LIN {X 0,Y 137.827,Z 379.001,A -85,B 0,C 180,E1 -25699.087,E2 -25699.087} C_VEL
LIN {X 0,Y 133.613,Z 369.148,A -85,B 0,C 180,E1 -25701.525,E2 -25701.525} C_VEL
LIN {X 0,Y 127.803,Z 359.632,A -85,B 0,C 180,E1 -25704.98,E2 -25704.98} C_VEL
LIN {X 0,Y 124.55,Z 355.02,A -85,B 0,C 180,E1 -25707.103,E2 -25707.103} C_VEL
LIN {X 0,Y 121.893,Z 351.23,A -85,B 0,C 180,E1 -25709.002,E2 -25709.002} C_VEL
LIN {X 0,Y 119.524,Z 348.351,A -85,B 0,C 180,E1 -25710.791,E2 -25710.791} C_VEL
LIN {X 0,Y 118.503,Z 346.486,A -85,B 0,C 180,E1 -25711.675,E2 -25711.675} C_VEL
LIN {X 0,Y 116.133,Z 344.433,A -85,B 0,C 180,E1 -25713.613,E2 -25713.613} C_VEL
LIN {X 0,Y 115.029,Z 342.02,A -85,B 0,C 180,E1 -25714.749,E2 -25714.749} C_VEL
LIN {X 0,Y 114.889,Z 341.174,A -85,B 0,C 180,E1 -25715.069,E2 -25715.069} C_VEL
LIN {X 0,Y 114.953,Z 341.137,A -85,B 0,C 180,E1 -25718.479,E2 -25718.479} C_VEL
LIN {X 0,Y 115.104,Z 341.145,A -85,B 0,C 180,E1 -25725.863,E2 -25725.863} C_VEL
LIN {X 0,Y 115.312,Z 341.081,A -85,B 0,C 180,E1 -25729.464,E2 -25729.464} C_VEL
LIN {X 0,Y 115.511,Z 341.094,A -85,B 0,C 180,E1 -25736.511,E2 -25736.511} C_VEL
LIN {X 0,Y 115.983,Z 341.003,A -85,B 0,C 180,E1 -25739.999,E2 -25739.999} C_VEL
LIN {X 0,Y 115.359,Z 341.105,A -85,B 0,C 180,E1 -25746.998,E2 -25746.998} C_VEL
LIN {X 0,Y 115.21,Z 341.099,A -85,B 0,C 180,E1 -25752.558,E2 -25752.558} C_VEL
LIN {X 0,Y 114.973,Z 341.127,A -85,B 0,C 180,E1 -25757.796,E2 -25757.796} C_VEL
LIN {X 0,Y 114.926,Z 341.156,A -85,B 0,C 180,E1 -25763.461,E2 -25763.461} C_VEL
LIN {X 0,Y 114.858,Z 341.154,A -85,B 0,C 180,E1 -25771.054,E2 -25771.054} C_VEL
LIN {X 0,Y 114.778,Z 341.146,A -85,B 0,C 180,E1 -25777.756,E2 -25777.756} C_VEL
LIN {X 0,Y 114.822,Z 341.142,A -85,B 0,C 180,E1 -25779.421,E2 -25779.421} C_VEL
LIN {X 0,Y 115.614,Z 343.676,A -85,B 0,C 180,E1 -25780.373,E2 -25780.373} C_VEL
LIN {X 0,Y 117.731,Z 346.081,A -85,B 0,C 180,E1 -25782.211,E2 -25782.211} C_VEL
LIN {X 0,Y 118.812,Z 346.913,A -85,B 0,C 180,E1 -25783.051,E2 -25783.051} C_VEL
LIN {X 0,Y 120.793,Z 350.186,A -85,B 0,C 180,E1 -25784.683,E2 -25784.683} C_VEL
LIN {X 0,Y 122.393,Z 351.931,A -85,B 0,C 180,E1 -25785.836,E2 -25785.836} C_VEL
LIN {X 0,Y 125.131,Z 355.737,A -85,B 0,C 180,E1 -25787.75,E2 -25787.75} C_VEL
LIN {X 0,Y 131.366,Z 365.259,A -85,B 0,C 180,E1 -25791.647,E2 -25791.647} C_VEL
LIN {X 0,Y 135.538,Z 372.511,A -85,B 0,C 180,E1 -25793.998,E2 -25793.998} C_VEL
LIN {X 0,Y 140.144,Z 381.658,A -85,B 0,C 180,E1 -25796.428,E2 -25796.428} C_VEL
LIN {X 0,Y 143.275,Z 388.687,A -85,B 0,C 180,E1 -25797.995,E2 -25797.995} C_VEL
LIN {X 0,Y 142.115,Z 408.083,A -85,B 0,C 180,E1 -25798.87,E2 -25798.87} C_VEL
LIN {X 0,Y 139.875,Z 437.734,A -85,B 0,C 180,E1 -25800.177,E2 -25800.177} C_VEL
LIN {X 0,Y 138.032,Z 451.323,A -85,B 0,C 180,E1 -25801.289,E2 -25801.289} C_VEL
LIN {X 0,Y 135.673,Z 463.657,A -85,B 0,C 180,E1 -25802.836,E2 -25802.836} C_VEL
LIN {X 0,Y 132.815,Z 475.522,A -85,B 0,C 180,E1 -25804.952,E2 -25804.952} C_VEL
LIN {X 0,Y 129.446,Z 486.941,A -85,B 0,C 180,E1 -25807.66,E2 -25807.66} C_VEL
LIN {X 0,Y 125.81,Z 497.272,A -85,B 0,C 180,E1 -25810.838,E2 -25810.838} C_VEL
LIN {X 0,Y 121.985,Z 507.34,A -85,B 0,C 180,E1 -25814.971,E2 -25814.971} C_VEL
LIN {X 0,Y 118.496,Z 516.2,A -85,B 0,C 180,E1 -25819.748,E2 -25819.748} C_VEL
LIN {X 0,Y 115.779,Z 523.275,A -85,B 0,C 180,E1 -25824.773,E2 -25824.773} C_VEL
LIN {X 0,Y 113.838,Z 528.929,A -85,B 0,C 180,E1 -25829.997,E2 -25829.997} C_VEL
LIN {X 0,Y 112.806,Z 532.82,A -85,B 0,C 180,E1 -25834.575,E2 -25834.575} C_VEL
LIN {X 0,Y 111.862,Z 536.768,A -85,B 0,C 180,E1 -25840.861,E2 -25840.861} C_VEL
LIN {X 0,Y 111.797,Z 538.454,A -85,B 0,C 180,E1 -25844.56,E2 -25844.56} C_VEL
LIN {X 0,Y 112.379,Z 540.208,A -85,B 0,C 180,E1 -25850.271,E2 -25850.271} C_VEL
LIN {X 0,Y 113.544,Z 540.951,A -85,B 0,C 180,E1 -25855.672,E2 -25855.672} C_VEL
LIN {X 0,Y 116.294,Z 540.626,A -85,B 0,C 180,E1 -25862.216,E2 -25862.216} C_VEL
LIN {X 0,Y 118.676,Z 539.642,A -85,B 0,C 180,E1 -25866.309,E2 -25866.309} C_VEL
LIN {X 0,Y 123.502,Z 536.925,A -85,B 0,C 180,E1 -25872.289,E2 -25872.289} C_VEL
LIN {X 0,Y 129.003,Z 533.061,A -85,B 0,C 180,E1 -25877.342,E2 -25877.342} C_VEL
LIN {X 0,Y 134.673,Z 528.328,A -85,B 0,C 180,E1 -25881.511,E2 -25881.511} C_VEL
LIN {X 0,Y 140.964,Z 522.244,A -85,B 0,C 180,E1 -25885.345,E2 -25885.345} C_VEL
LIN {X 0,Y 147.922,Z 514.608,A -85,B 0,C 180,E1 -25888.777,E2 -25888.777} C_VEL
LIN {X 0,Y 154.047,Z 506.758,A -85,B 0,C 180,E1 -25891.424,E2 -25891.424} C_VEL
LIN {X 0,Y 160.683,Z 496.79,A -85,B 0,C 180,E1 -25893.929,E2 -25893.929} C_VEL
LIN {X 0,Y 166.481,Z 486.303,A -85,B 0,C 180,E1 -25895.903,E2 -25895.903} C_VEL
LIN {X 0,Y 171.312,Z 475.836,A -85,B 0,C 180,E1 -25897.37,E2 -25897.37} C_VEL
LIN {X 0,Y 175.536,Z 464.261,A -85,B 0,C 180,E1 -25898.628,E2 -25898.628} C_VEL
LIN {X 0,Y 178.99,Z 451.384,A -85,B 0,C 180,E1 -25899.64,E2 -25899.64} C_VEL
LIN {X 0,Y 181.472,Z 437.921,A -85,B 0,C 180,E1 -25900.311,E2 -25900.311} C_VEL
LIN {X 0,Y 183.082,Z 422.653,A -85,B 0,C 180,E1 -25900.76,E2 -25900.76} C_VEL
LIN {X 0,Y 179.542,Z 415.553,A -85,B 0,C 180,E1 -25903.806,E2 -25903.806} C_VEL
LIN {X 0,Y 176.526,Z 410.032,A -85,B 0,C 180,E1 -25906.785,E2 -25906.785} C_VEL
LIN {X 0,Y 174.132,Z 405.888,A -85,B 0,C 180,E1 -25909.54,E2 -25909.54} C_VEL
LIN {X 0,Y 172.909,Z 403.751,A -85,B 0,C 180,E1 -25911.158,E2 -25911.158} C_VEL
LIN {X 0,Y 170.704,Z 399.785,A -85,B 0,C 180,E1 -25914.759,E2 -25914.759} C_VEL
LIN {X 0,Y 168.841,Z 396.541,A -85,B 0,C 180,E1 -25919.062,E2 -25919.062} C_VEL
LIN {X 0,Y 168.584,Z 395.7,A -85,B 0,C 180,E1 -25920.001,E2 -25920.001} C_VEL
LIN {X 0,Y 167.507,Z 395.197,A -85,B 0,C 180,E1 -25924.814,E2 -25924.814} C_VEL
LIN {X 0,Y 167.607,Z 395.272,A -85,B 0,C 180,E1 -25929.656,E2 -25929.656} C_VEL
LIN {X 0,Y 168.546,Z 396.155,A -85,B 0,C 180,E1 -25933.716,E2 -25933.716} C_VEL
LIN {X 0,Y 170.103,Z 399.496,A -85,B 0,C 180,E1 -25937.876,E2 -25937.876} C_VEL
LIN {X 0,Y 171.176,Z 400.958,A -85,B 0,C 180,E1 -25939.832,E2 -25939.832} C_VEL
LIN {X 0,Y 173.514,Z 405.486,A -85,B 0,C 180,E1 -25943.419,E2 -25943.419} C_VEL
LIN {X 0,Y 175.851,Z 410.567,A -85,B 0,C 180,E1 -25946.348,E2 -25946.348} C_VEL
LIN {X 0,Y 178.897,Z 417.775,A -85,B 0,C 180,E1 -25949.606,E2 -25949.606} C_VEL
LIN {X 0,Y 181.846,Z 425.459,A -85,B 0,C 180,E1 -25952.37,E2 -25952.37} C_VEL
LIN {X 0,Y 182.641,Z 427.679,A -85,B 0,C 180,E1 -25953.068,E2 -25953.068} C_VEL
LIN {X 0,Y 180.767,Z 445.11,A -85,B 0,C 180,E1 -25953.661,E2 -25953.661} C_VEL
LIN {X 0,Y 178.134,Z 458.354,A -85,B 0,C 180,E1 -25954.359,E2 -25954.359} C_VEL
LIN {X 0,Y 174.747,Z 469.708,A -85,B 0,C 180,E1 -25955.168,E2 -25955.168} C_VEL
LIN {X 0,Y 170.165,Z 481.545,A -85,B 0,C 180,E1 -25956.358,E2 -25956.358} C_VEL
LIN {X 0,Y 164.843,Z 492.752,A -85,B 0,C 180,E1 -25957.936,E2 -25957.936} C_VEL
LIN {X 0,Y 158.973,Z 502.9,A -85,B 0,C 180,E1 -25959.818,E2 -25959.818} C_VEL
LIN {X 0,Y 153.372,Z 511.22,A -85,B 0,C 180,E1 -25961.877,E2 -25961.877} C_VEL
LIN {X 0,Y 146.218,Z 520.28,A -85,B 0,C 180,E1 -25964.853,E2 -25964.853} C_VEL
LIN {X 0,Y 139.495,Z 527.609,A -85,B 0,C 180,E1 -25968.125,E2 -25968.125} C_VEL
LIN {X 0,Y 134.368,Z 532.602,A -85,B 0,C 180,E1 -25971.127,E2 -25971.127} C_VEL
LIN {X 0,Y 129.267,Z 537.189,A -85,B 0,C 180,E1 -25974.823,E2 -25974.823} C_VEL
LIN {X 0,Y 124.031,Z 541.242,A -85,B 0,C 180,E1 -25979.342,E2 -25979.342} C_VEL
LIN {X 0,Y 118.724,Z 544.762,A -85,B 0,C 180,E1 -25985.524,E2 -25985.524} C_VEL
LIN {X 0,Y 116.569,Z 545.891,A -85,B 0,C 180,E1 -25988.796,E2 -25988.796} C_VEL
LIN {X 0,Y 113.713,Z 546.98,A -85,B 0,C 180,E1 -25995.69,E2 -25995.69} C_VEL
LIN {X 0,Y 112.862,Z 546.963,A -85,B 0,C 180,E1 -25999.237,E2 -25999.237} C_VEL
LIN {X 0,Y 112.354,Z 546.555,A -85,B 0,C 180,E1 -26002.817,E2 -26002.817} C_VEL
LIN {X 0,Y 112.262,Z 545.725,A -85,B 0,C 180,E1 -26006.414,E2 -26006.414} C_VEL
LIN {X 0,Y 112.334,Z 544.497,A -85,B 0,C 180,E1 -26010.003,E2 -26010.003} C_VEL
LIN {X 0,Y 112.247,Z 541.82,A -85,B 0,C 180,E1 -26015.392,E2 -26015.392} C_VEL
LIN {X 0,Y 112.798,Z 538.095,A -85,B 0,C 180,E1 -26020.776,E2 -26020.776} C_VEL
LIN {X 0,Y 113.999,Z 533.213,A -85,B 0,C 180,E1 -26026.11,E2 -26026.11} C_VEL
LIN {X 0,Y 116.159,Z 527.043,A -85,B 0,C 180,E1 -26031.289,E2 -26031.289} C_VEL
LIN {X 0,Y 119.107,Z 519.342,A -85,B 0,C 180,E1 -26036.269,E2 -26036.269} C_VEL
LIN {X 0,Y 122.141,Z 511.23,A -85,B 0,C 180,E1 -26040.332,E2 -26040.332} C_VEL
LIN {X 0,Y 125.723,Z 501.735,A -85,B 0,C 180,E1 -26043.99,E2 -26043.99} C_VEL
LIN {X 0,Y 129.315,Z 490.95,A -85,B 0,C 180,E1 -26047.205,E2 -26047.205} C_VEL
LIN {X 0,Y 132.655,Z 480.586,A -85,B 0,C 180,E1 -26049.479,E2 -26049.479} C_VEL
LIN {X 0,Y 133.738,Z 476.295,A -85,B 0,C 180,E1 -26050.286,E2 -26050.286} C_VEL
LIN {X 0,Y 134.047,Z 472.751,A -85,B 0,C 180,E1 -26051.07,E2 -26051.07} C_VEL
LIN {X 0,Y 132.999,Z 467.14,A -85,B 0,C 180,E1 -26052.639,E2 -26052.639} C_VEL
LIN {X 0,Y 131.908,Z 461.392,A -85,B 0,C 180,E1 -26054.093,E2 -26054.093} C_VEL
LIN {X 0,Y 132.097,Z 457.639,A -85,B 0,C 180,E1 -26054.66,E2 -26054.66} C_VEL
LIN {X 0,Y 134.126,Z 443.975,A -85,B 0,C 180,E1 -26055.786,E2 -26055.786} C_VEL
LIN {X 0,Y 137.136,Z 402.806,A -85,B 0,C 180,E1 -26057.681,E2 -26057.681} C_VEL
LIN {X 0,Y 137.217,Z 397.25,A -85,B 0,C 180,E1 -26058.038,E2 -26058.038} C_VEL
LIN {X 0,Y 136.74,Z 393.549,A -85,B 0,C 180,E1 -26058.476,E2 -26058.476} C_VEL
LIN {X 0,Y 132.767,Z 381.798,A -85,B 0,C 180,E1 -26060.93,E2 -26060.93} C_VEL
LIN {X 0,Y 129.383,Z 373.685,A -85,B 0,C 180,E1 -26063.064,E2 -26063.064} C_VEL
LIN {X 0,Y 123.95,Z 364.6,A -85,B 0,C 180,E1 -26066.572,E2 -26066.572} C_VEL
LIN {X 0,Y 118.97,Z 357.189,A -85,B 0,C 180,E1 -26070.254,E2 -26070.254} C_VEL
LIN {X 0,Y 116.317,Z 353.693,A -85,B 0,C 180,E1 -26072.444,E2 -26072.444} C_VEL
LIN {X 0,Y 115.584,Z 352.531,A -85,B 0,C 180,E1 -26073.112,E2 -26073.112} C_VEL
LIN {X 0,Y 113.146,Z 349.883,A -85,B 0,C 180,E1 -26075.342,E2 -26075.342} C_VEL
LIN {X 0,Y 112.083,Z 347.678,A -85,B 0,C 180,E1 -26076.525,E2 -26076.525} C_VEL
LIN {X 0,Y 109.323,Z 345.51,A -85,B 0,C 180,E1 -26079.416,E2 -26079.416} C_VEL
LIN {X 0,Y 108.116,Z 343.183,A -85,B 0,C 180,E1 -26081.032,E2 -26081.032} C_VEL
LIN {X 0,Y 107.892,Z 342.014,A -85,B 0,C 180,E1 -26081.484,E2 -26081.484} C_VEL
LIN {X 0,Y 108.212,Z 341.969,A -85,B 0,C 180,E1 -26088.764,E2 -26088.764} C_VEL
LIN {X 0,Y 108.296,Z 341.957,A -85,B 0,C 180,E1 -26092.542,E2 -26092.542} C_VEL
LIN {X 0,Y 108.909,Z 341.882,A -85,B 0,C 180,E1 -26099.999,E2 -26099.999} C_VEL
LIN {X 0,Y 108.298,Z 341.987,A -85,B 0,C 180,E1 -26107.457,E2 -26107.457} C_VEL
LIN {X 0,Y 108.144,Z 341.974,A -85,B 0,C 180,E1 -26112.873,E2 -26112.873} C_VEL
LIN {X 0,Y 107.872,Z 342.025,A -85,B 0,C 180,E1 -26119.01,E2 -26119.01} C_VEL
LIN {X 0,Y 107.833,Z 342.028,A -85,B 0,C 180,E1 -26124.147,E2 -26124.147} C_VEL
LIN {X 0,Y 107.765,Z 342.055,A -85,B 0,C 180,E1 -26132.742,E2 -26132.742} C_VEL
LIN {X 0,Y 108.751,Z 344.913,A -85,B 0,C 180,E1 -26134.366,E2 -26134.366} C_VEL
LIN {X 0,Y 110.78,Z 347.032,A -85,B 0,C 180,E1 -26136.674,E2 -26136.674} C_VEL
LIN {X 0,Y 112.145,Z 347.931,A -85,B 0,C 180,E1 -26138.028,E2 -26138.028} C_VEL
LIN {X 0,Y 113.954,Z 351.053,A -85,B 0,C 180,E1 -26139.925,E2 -26139.925} C_VEL
LIN {X 0,Y 116.048,Z 353.188,A -85,B 0,C 180,E1 -26141.771,E2 -26141.771} C_VEL
LIN {X 0,Y 118.459,Z 356.701,A -85,B 0,C 180,E1 -26143.827,E2 -26143.827} C_VEL
LIN {X 0,Y 119.687,Z 358.436,A -85,B 0,C 180,E1 -26144.799,E2 -26144.799} C_VEL
LIN {X 0,Y 123.602,Z 364.137,A -85,B 0,C 180,E1 -26147.66,E2 -26147.66} C_VEL
LIN {X 0,Y 128.584,Z 372.074,A -85,B 0,C 180,E1 -26150.898,E2 -26150.898} C_VEL
LIN {X 0,Y 134.41,Z 383.213,A -85,B 0,C 180,E1 -26154.323,E2 -26154.323} C_VEL
LIN {X 0,Y 137.862,Z 391.022,A -85,B 0,C 180,E1 -26156.231,E2 -26156.231} C_VEL
LIN {X 0,Y 134.356,Z 437.827,A -85,B 0,C 180,E1 -26158.318,E2 -26158.318} C_VEL
LIN {X 0,Y 132.383,Z 451.784,A -85,B 0,C 180,E1 -26159.489,E2 -26159.489} C_VEL
LIN {X 0,Y 129.88,Z 464.097,A -85,B 0,C 180,E1 -26161.075,E2 -26161.075} C_VEL
LIN {X 0,Y 126.877,Z 475.904,A -85,B 0,C 180,E1 -26163.249,E2 -26163.249} C_VEL
LIN {X 0,Y 123.326,Z 487.32,A -85,B 0,C 180,E1 -26166.052,E2 -26166.052} C_VEL
LIN {X 0,Y 119.5,Z 497.588,A -85,B 0,C 180,E1 -26169.334,E2 -26169.334} C_VEL
LIN {X 0,Y 115.821,Z 506.81,A -85,B 0,C 180,E1 -26173.245,E2 -26173.245} C_VEL
LIN {X 0,Y 112.034,Z 515.794,A -85,B 0,C 180,E1 -26178.233,E2 -26178.233} C_VEL
LIN {X 0,Y 109.056,Z 523.018,A -85,B 0,C 180,E1 -26183.521,E2 -26183.521} C_VEL
LIN {X 0,Y 107.232,Z 527.89,A -85,B 0,C 180,E1 -26188.119,E2 -26188.119} C_VEL
LIN {X 0,Y 105.721,Z 533.01,A -85,B 0,C 180,E1 -26194.334,E2 -26194.334} C_VEL
LIN {X 0,Y 104.888,Z 536.261,A -85,B 0,C 180,E1 -26199.64,E2 -26199.64} C_VEL
LIN {X 0,Y 104.732,Z 538.867,A -85,B 0,C 180,E1 -26205.567,E2 -26205.567} C_VEL
LIN {X 0,Y 105.375,Z 540.383,A -85,B 0,C 180,E1 -26210.978,E2 -26210.978} C_VEL
LIN {X 0,Y 106.907,Z 541.182,A -85,B 0,C 180,E1 -26217.394,E2 -26217.394} C_VEL
LIN {X 0,Y 109.666,Z 540.852,A -85,B 0,C 180,E1 -26223.582,E2 -26223.582} C_VEL
LIN {X 0,Y 112.772,Z 539.685,A -85,B 0,C 180,E1 -26228.546,E2 -26228.546} C_VEL
LIN {X 0,Y 117.499,Z 537.203,A -85,B 0,C 180,E1 -26234.131,E2 -26234.131} C_VEL
LIN {X 0,Y 122.194,Z 534.189,A -85,B 0,C 180,E1 -26238.386,E2 -26238.386} C_VEL
LIN {X 0,Y 128.546,Z 529.387,A -85,B 0,C 180,E1 -26243.03,E2 -26243.03} C_VEL
LIN {X 0,Y 135.72,Z 522.973,A -85,B 0,C 180,E1 -26247.291,E2 -26247.291} C_VEL
LIN {X 0,Y 142.801,Z 515.651,A -85,B 0,C 180,E1 -26250.67,E2 -26250.67} C_VEL
LIN {X 0,Y 149.335,Z 507.74,A -85,B 0,C 180,E1 -26253.397,E2 -26253.397} C_VEL
LIN {X 0,Y 156.111,Z 498.172,A -85,B 0,C 180,E1 -26255.846,E2 -26255.846} C_VEL
LIN {X 0,Y 162.206,Z 487.75,A -85,B 0,C 180,E1 -26257.832,E2 -26257.832} C_VEL
LIN {X 0,Y 167.172,Z 477.558,A -85,B 0,C 180,E1 -26259.286,E2 -26259.286} C_VEL
LIN {X 0,Y 172.029,Z 464.986,A -85,B 0,C 180,E1 -26260.649,E2 -26260.649} C_VEL
LIN {X 0,Y 175.423,Z 453.15,A -85,B 0,C 180,E1 -26261.583,E2 -26261.583} C_VEL
LIN {X 0,Y 178.092,Z 439.722,A -85,B 0,C 180,E1 -26262.267,E2 -26262.267} C_VEL
LIN {X 0,Y 179.652,Z 426.224,A -85,B 0,C 180,E1 -26262.69,E2 -26262.69} C_VEL
LIN {X 0,Y 176.367,Z 419.516,A -85,B 0,C 180,E1 -26265.851,E2 -26265.851} C_VEL
LIN {X 0,Y 173.495,Z 414.015,A -85,B 0,C 180,E1 -26269.106,E2 -26269.106} C_VEL
LIN {X 0,Y 171.402,Z 410.289,A -85,B 0,C 180,E1 -26271.942,E2 -26271.942} C_VEL
LIN {X 0,Y 169.34,Z 406.418,A -85,B 0,C 180,E1 -26275.593,E2 -26275.593} C_VEL
LIN {X 0,Y 167.703,Z 403.164,A -85,B 0,C 180,E1 -26279.843,E2 -26279.843} C_VEL
LIN {X 0,Y 167.333,Z 402.501,A -85,B 0,C 180,E1 -26281.204,E2 -26281.204} C_VEL
LIN {X 0,Y 166.57,Z 402.195,A -85,B 0,C 180,E1 -26288.143,E2 -26288.143} C_VEL
LIN {X 0,Y 167.549,Z 403.229,A -85,B 0,C 180,E1 -26293.411,E2 -26293.411} C_VEL
LIN {X 0,Y 169.1,Z 406.549,A -85,B 0,C 180,E1 -26297.693,E2 -26297.693} C_VEL
LIN {X 0,Y 169.95,Z 407.804,A -85,B 0,C 180,E1 -26299.32,E2 -26299.32} C_VEL
LIN {X 0,Y 171.934,Z 412,A -85,B 0,C 180,E1 -26302.613,E2 -26302.613} C_VEL
LIN {X 0,Y 173.992,Z 416.742,A -85,B 0,C 180,E1 -26305.389,E2 -26305.389} C_VEL
LIN {X 0,Y 176.855,Z 424.029,A -85,B 0,C 180,E1 -26308.693,E2 -26308.693} C_VEL
LIN {X 0,Y 179.269,Z 430.9,A -85,B 0,C 180,E1 -26311.154,E2 -26311.154} C_VEL
LIN {X 0,Y 177.459,Z 446.068,A -85,B 0,C 180,E1 -26311.672,E2 -26311.672} C_VEL
LIN {X 0,Y 174.693,Z 458.981,A -85,B 0,C 180,E1 -26312.35,E2 -26312.35} C_VEL
LIN {X 0,Y 170.9,Z 470.992,A -85,B 0,C 180,E1 -26313.208,E2 -26313.208} C_VEL
LIN {X 0,Y 166.094,Z 482.776,A -85,B 0,C 180,E1 -26314.405,E2 -26314.405} C_VEL
LIN {X 0,Y 160.613,Z 493.71,A -85,B 0,C 180,E1 -26315.956,E2 -26315.956} C_VEL
LIN {X 0,Y 153.902,Z 504.561,A -85,B 0,C 180,E1 -26318.031,E2 -26318.031} C_VEL
LIN {X 0,Y 147.469,Z 513.386,A -85,B 0,C 180,E1 -26320.317,E2 -26320.317} C_VEL
LIN {X 0,Y 140.126,Z 522.031,A -85,B 0,C 180,E1 -26323.348,E2 -26323.348} C_VEL
LIN {X 0,Y 133.195,Z 528.957,A -85,B 0,C 180,E1 -26326.695,E2 -26326.695} C_VEL
LIN {X 0,Y 126.915,Z 534.525,A -85,B 0,C 180,E1 -26330.449,E2 -26330.449} C_VEL
LIN {X 0,Y 121.385,Z 538.929,A -85,B 0,C 180,E1 -26334.625,E2 -26334.625} C_VEL
LIN {X 0,Y 117.978,Z 541.271,A -85,B 0,C 180,E1 -26337.583,E2 -26337.583} C_VEL
LIN {X 0,Y 114.95,Z 543.196,A -85,B 0,C 180,E1 -26340.721,E2 -26340.721} C_VEL
LIN {X 0,Y 112.281,Z 544.703,A -85,B 0,C 180,E1 -26344.018,E2 -26344.018} C_VEL
LIN {X 0,Y 109.958,Z 545.777,A -85,B 0,C 180,E1 -26347.454,E2 -26347.454} C_VEL
LIN {X 0,Y 106.835,Z 546.798,A -85,B 0,C 180,E1 -26354.748,E2 -26354.748} C_VEL
LIN {X 0,Y 105.872,Z 546.744,A -85,B 0,C 180,E1 -26358.517,E2 -26358.517} C_VEL
LIN {X 0,Y 105.18,Z 545.406,A -85,B 0,C 180,E1 -26366.172,E2 -26366.172} C_VEL
LIN {X 0,Y 105.235,Z 544.142,A -85,B 0,C 180,E1 -26370.003,E2 -26370.003} C_VEL
LIN {X 0,Y 105.191,Z 541.393,A -85,B 0,C 180,E1 -26375.755,E2 -26375.755} C_VEL
LIN {X 0,Y 105.807,Z 537.588,A -85,B 0,C 180,E1 -26381.498,E2 -26381.498} C_VEL
LIN {X 0,Y 107.157,Z 532.622,A -85,B 0,C 180,E1 -26387.169,E2 -26387.169} C_VEL
LIN {X 0,Y 109.555,Z 526.362,A -85,B 0,C 180,E1 -26392.641,E2 -26392.641} C_VEL
LIN {X 0,Y 112.767,Z 518.513,A -85,B 0,C 180,E1 -26397.871,E2 -26397.871} C_VEL
LIN {X 0,Y 115.591,Z 511.301,A -85,B 0,C 180,E1 -26401.655,E2 -26401.655} C_VEL
LIN {X 0,Y 119.436,Z 501.688,A -85,B 0,C 180,E1 -26405.53,E2 -26405.53} C_VEL
LIN {X 0,Y 123.233,Z 490.936,A -85,B 0,C 180,E1 -26408.857,E2 -26408.857} C_VEL
LIN {X 0,Y 126.729,Z 480.615,A -85,B 0,C 180,E1 -26411.193,E2 -26411.193} C_VEL
LIN {X 0,Y 129.716,Z 469.364,A -85,B 0,C 180,E1 -26413.162,E2 -26413.162} C_VEL
LIN {X 0,Y 132.097,Z 457.639,A -85,B 0,C 180,E1 -26414.66,E2 -26414.66} C_VEL
LIN {X 0,Y 132.65,Z 451.966,A -85,B 0,C 180,E1 -26415.339,E2 -26415.339} C_VEL
LIN {X 0,Y 131.699,Z 442.685,A -85,B 0,C 180,E1 -26416.8,E2 -26416.8} C_VEL
LIN {X 0,Y 130.256,Z 433.312,A -85,B 0,C 180,E1 -26418.129,E2 -26418.129} C_VEL
LIN {X 0,Y 130.131,Z 427.483,A -85,B 0,C 180,E1 -26418.599,E2 -26418.599} C_VEL
LIN {X 0,Y 132.016,Z 399.817,A -85,B 0,C 180,E1 -26419.892,E2 -26419.892} C_VEL
LIN {X 0,Y 131.718,Z 396.296,A -85,B 0,C 180,E1 -26420.28,E2 -26420.28} C_VEL
LIN {X 0,Y 128.179,Z 385.527,A -85,B 0,C 180,E1 -26422.674,E2 -26422.674} C_VEL
LIN {X 0,Y 125.232,Z 378.127,A -85,B 0,C 180,E1 -26424.714,E2 -26424.714} C_VEL
LIN {X 0,Y 120.22,Z 369.561,A -85,B 0,C 180,E1 -26428.254,E2 -26428.254} C_VEL
LIN {X 0,Y 115.921,Z 362.893,A -85,B 0,C 180,E1 -26431.727,E2 -26431.727} C_VEL
LIN {X 0,Y 113.232,Z 359.07,A -85,B 0,C 180,E1 -26434.17,E2 -26434.17} C_VEL
LIN {X 0,Y 110.226,Z 355.254,A -85,B 0,C 180,E1 -26437.212,E2 -26437.212} C_VEL
LIN {X 0,Y 109.479,Z 353.942,A -85,B 0,C 180,E1 -26438.09,E2 -26438.09} C_VEL
LIN {X 0,Y 106.783,Z 351.205,A -85,B 0,C 180,E1 -26441.285,E2 -26441.285} C_VEL
LIN {X 0,Y 105.597,Z 348.724,A -85,B 0,C 180,E1 -26443.071,E2 -26443.071} C_VEL
LIN {X 0,Y 103.163,Z 347.119,A -85,B 0,C 180,E1 -26446.64,E2 -26446.64} C_VEL
LIN {X 0,Y 101.442,Z 344.121,A -85,B 0,C 180,E1 -26450.151,E2 -26450.151} C_VEL
LIN {X 0,Y 101.182,Z 342.836,A -85,B 0,C 180,E1 -26451.134,E2 -26451.134} C_VEL
LIN {X 0,Y 101.836,Z 342.761,A -85,B 0,C 180,E1 -26459.999,E2 -26459.999} C_VEL
LIN {X 0,Y 101.234,Z 342.871,A -85,B 0,C 180,E1 -26467.98,E2 -26467.98} C_VEL
LIN {X 0,Y 101.056,Z 342.852,A -85,B 0,C 180,E1 -26473.171,E2 -26473.171} C_VEL
LIN {X 0,Y 100.877,Z 343.022,A -85,B 0,C 180,E1 -26482.935,E2 -26482.935} C_VEL
LIN {X 0,Y 101.554,Z 345.434,A -85,B 0,C 180,E1 -26484.835,E2 -26484.835} C_VEL
LIN {X 0,Y 103.611,Z 347.831,A -85,B 0,C 180,E1 -26488.623,E2 -26488.623} C_VEL
LIN {X 0,Y 105.558,Z 348.891,A -85,B 0,C 180,E1 -26491.378,E2 -26491.378} C_VEL
LIN {X 0,Y 107.009,Z 351.782,A -85,B 0,C 180,E1 -26493.521,E2 -26493.521} C_VEL
LIN {X 0,Y 109.465,Z 354.023,A -85,B 0,C 180,E1 -26496.372,E2 -26496.372} C_VEL
LIN {X 0,Y 112.395,Z 358.211,A -85,B 0,C 180,E1 -26499.514,E2 -26499.514} C_VEL
LIN {X 0,Y 113.497,Z 359.592,A -85,B 0,C 180,E1 -26500.564,E2 -26500.564} C_VEL
LIN {X 0,Y 116.716,Z 364.251,A -85,B 0,C 180,E1 -26503.434,E2 -26503.434} C_VEL
LIN {X 0,Y 121.242,Z 371.145,A -85,B 0,C 180,E1 -26506.964,E2 -26506.964} C_VEL
LIN {X 0,Y 125.992,Z 379.412,A -85,B 0,C 180,E1 -26510.243,E2 -26510.243} C_VEL
LIN {X 0,Y 131.022,Z 389.808,A -85,B 0,C 180,E1 -26513.394,E2 -26513.394} C_VEL
LIN {X 0,Y 132.563,Z 393.469,A -85,B 0,C 180,E1 -26514.322,E2 -26514.322} C_VEL
LIN {X 0,Y 128.973,Z 438.09,A -85,B 0,C 180,E1 -26516.315,E2 -26516.315} C_VEL
LIN {X 0,Y 126.971,Z 451.583,A -85,B 0,C 180,E1 -26517.453,E2 -26517.453} C_VEL
LIN {X 0,Y 124.222,Z 464.53,A -85,B 0,C 180,E1 -26519.151,E2 -26519.151} C_VEL
LIN {X 0,Y 121.061,Z 476.286,A -85,B 0,C 180,E1 -26521.381,E2 -26521.381} C_VEL
LIN {X 0,Y 117.247,Z 487.838,A -85,B 0,C 180,E1 -26524.312,E2 -26524.312} C_VEL
LIN {X 0,Y 113.283,Z 497.901,A -85,B 0,C 180,E1 -26527.663,E2 -26527.663} C_VEL
LIN {X 0,Y 108.996,Z 507.926,A -85,B 0,C 180,E1 -26532.162,E2 -26532.162} C_VEL
LIN {X 0,Y 105.052,Z 516.753,A -85,B 0,C 180,E1 -26537.439,E2 -26537.439} C_VEL
LIN {X 0,Y 101.98,Z 523.789,A -85,B 0,C 180,E1 -26543.07,E2 -26543.07} C_VEL
LIN {X 0,Y 99.538,Z 530.237,A -85,B 0,C 180,E1 -26549.996,E2 -26549.996} C_VEL
LIN {X 0,Y 98.226,Z 534.494,A -85,B 0,C 180,E1 -26556.157,E2 -26556.157} C_VEL
LIN {X 0,Y 97.602,Z 537.687,A -85,B 0,C 180,E1 -26562.471,E2 -26562.471} C_VEL
LIN {X 0,Y 97.712,Z 539.275,A -85,B 0,C 180,E1 -26566.716,E2 -26566.716} C_VEL
LIN {X 0,Y 98.369,Z 540.552,A -85,B 0,C 180,E1 -26571.756,E2 -26571.756} C_VEL
LIN {X 0,Y 100.376,Z 541.412,A -85,B 0,C 180,E1 -26579.344,E2 -26579.344} C_VEL
LIN {X 0,Y 103.118,Z 541.078,A -85,B 0,C 180,E1 -26585.13,E2 -26585.13} C_VEL
LIN {X 0,Y 107.037,Z 539.732,A -85,B 0,C 180,E1 -26591.036,E2 -26591.036} C_VEL
LIN {X 0,Y 111.625,Z 537.494,A -85,B 0,C 180,E1 -26596.168,E2 -26596.168} C_VEL
LIN {X 0,Y 117.392,Z 534.049,A -85,B 0,C 180,E1 -26601.098,E2 -26601.098} C_VEL
LIN {X 0,Y 124.254,Z 529.106,A -85,B 0,C 180,E1 -26605.804,E2 -26605.804} C_VEL
LIN {X 0,Y 131.84,Z 522.554,A -85,B 0,C 180,E1 -26610.018,E2 -26610.018} C_VEL
LIN {X 0,Y 139.762,Z 514.635,A -85,B 0,C 180,E1 -26613.506,E2 -26613.506} C_VEL
LIN {X 0,Y 146.171,Z 507.04,A -85,B 0,C 180,E1 -26615.991,E2 -26615.991} C_VEL
LIN {X 0,Y 153.101,Z 497.425,A -85,B 0,C 180,E1 -26618.319,E2 -26618.319} C_VEL
LIN {X 0,Y 159.57,Z 486.523,A -85,B 0,C 180,E1 -26620.284,E2 -26620.284} C_VEL
LIN {X 0,Y 164.718,Z 476.016,A -85,B 0,C 180,E1 -26621.675,E2 -26621.675} C_VEL
LIN {X 0,Y 169.161,Z 464.55,A -85,B 0,C 180,E1 -26622.846,E2 -26622.846} C_VEL
LIN {X 0,Y 172.774,Z 451.879,A -85,B 0,C 180,E1 -26623.793,E2 -26623.793} C_VEL
LIN {X 0,Y 175.335,Z 438.887,A -85,B 0,C 180,E1 -26624.409,E2 -26624.409} C_VEL
LIN {X 0,Y 176.4,Z 429.935,A -85,B 0,C 180,E1 -26624.704,E2 -26624.704} C_VEL
LIN {X 0,Y 173.367,Z 423.435,A -85,B 0,C 180,E1 -26628.028,E2 -26628.028} C_VEL
LIN {X 0,Y 170.679,Z 418.283,A -85,B 0,C 180,E1 -26631.561,E2 -26631.561} C_VEL
LIN {X 0,Y 168.136,Z 413.212,A -85,B 0,C 180,E1 -26636.182,E2 -26636.182} C_VEL
LIN {X 0,Y 166.603,Z 409.816,A -85,B 0,C 180,E1 -26640.605,E2 -26640.605} C_VEL
LIN {X 0,Y 166.154,Z 409.331,A -85,B 0,C 180,E1 -26642.425,E2 -26642.425} C_VEL
LIN {X 0,Y 165.694,Z 409.245,A -85,B 0,C 180,E1 -26648.186,E2 -26648.186} C_VEL
LIN {X 0,Y 166.492,Z 410.012,A -85,B 0,C 180,E1 -26652.786,E2 -26652.786} C_VEL
LIN {X 0,Y 167.88,Z 413.305,A -85,B 0,C 180,E1 -26657.041,E2 -26657.041} C_VEL
LIN {X 0,Y 168.749,Z 414.718,A -85,B 0,C 180,E1 -26658.831,E2 -26658.831} C_VEL
LIN {X 0,Y 170.393,Z 418.499,A -85,B 0,C 180,E1 -26661.791,E2 -26661.791} C_VEL
LIN {X 0,Y 172.502,Z 423.783,A -85,B 0,C 180,E1 -26664.844,E2 -26664.844} C_VEL
LIN {X 0,Y 175.175,Z 431.265,A -85,B 0,C 180,E1 -26668.128,E2 -26668.128} C_VEL
LIN {X 0,Y 176.091,Z 434.106,A -85,B 0,C 180,E1 -26669.158,E2 -26669.158} C_VEL
LIN {X 0,Y 174.215,Z 447.748,A -85,B 0,C 180,E1 -26669.635,E2 -26669.635} C_VEL
LIN {X 0,Y 171.04,Z 461.125,A -85,B 0,C 180,E1 -26670.363,E2 -26670.363} C_VEL
LIN {X 0,Y 167.262,Z 472.281,A -85,B 0,C 180,E1 -26671.161,E2 -26671.161} C_VEL
LIN {X 0,Y 162.226,Z 483.99,A -85,B 0,C 180,E1 -26672.356,E2 -26672.356} C_VEL
LIN {X 0,Y 156.57,Z 494.587,A -85,B 0,C 180,E1 -26673.864,E2 -26673.864} C_VEL
LIN {X 0,Y 149.649,Z 505.249,A -85,B 0,C 180,E1 -26675.898,E2 -26675.898} C_VEL
LIN {X 0,Y 142.994,Z 513.928,A -85,B 0,C 180,E1 -26678.156,E2 -26678.156} C_VEL
LIN {X 0,Y 135.37,Z 522.399,A -85,B 0,C 180,E1 -26681.171,E2 -26681.171} C_VEL
LIN {X 0,Y 128.139,Z 529.217,A -85,B 0,C 180,E1 -26684.524,E2 -26684.524} C_VEL
LIN {X 0,Y 121.51,Z 534.695,A -85,B 0,C 180,E1 -26688.311,E2 -26688.311} C_VEL
LIN {X 0,Y 115.658,Z 539.012,A -85,B 0,C 180,E1 -26692.584,E2 -26692.584} C_VEL
LIN {X 0,Y 112.051,Z 541.312,A -85,B 0,C 180,E1 -26695.637,E2 -26695.637} C_VEL
LIN {X 0,Y 108.787,Z 543.194,A -85,B 0,C 180,E1 -26698.885,E2 -26698.885} C_VEL
LIN {X 0,Y 103.419,Z 545.665,A -85,B 0,C 180,E1 -26705.941,E2 -26705.941} C_VEL
LIN {X 0,Y 99.98,Z 546.616,A -85,B 0,C 180,E1 -26713.673,E2 -26713.673} C_VEL
LIN {X 0,Y 98.915,Z 546.505,A -85,B 0,C 180,E1 -26717.697,E2 -26717.697} C_VEL
LIN {X 0,Y 98.091,Z 545.086,A -85,B 0,C 180,E1 -26725.895,E2 -26725.895} C_VEL
LIN {X 0,Y 98.147,Z 543.788,A -85,B 0,C 180,E1 -26730.004,E2 -26730.004} C_VEL
LIN {X 0,Y 98.115,Z 540.964,A -85,B 0,C 180,E1 -26736.172,E2 -26736.172} C_VEL
LIN {X 0,Y 98.812,Z 537.08,A -85,B 0,C 180,E1 -26742.324,E2 -26742.324} C_VEL
LIN {X 0,Y 100.338,Z 532.029,A -85,B 0,C 180,E1 -26748.376,E2 -26748.376} C_VEL
LIN {X 0,Y 102.976,Z 525.671,A -85,B 0,C 180,E1 -26754.177,E2 -26754.177} C_VEL
LIN {X 0,Y 106.518,Z 517.671,A -85,B 0,C 180,E1 -26759.663,E2 -26759.663} C_VEL
LIN {X 0,Y 109.132,Z 511.325,A -85,B 0,C 180,E1 -26763.154,E2 -26763.154} C_VEL
LIN {X 0,Y 113.252,Z 501.643,A -85,B 0,C 180,E1 -26767.236,E2 -26767.236} C_VEL
LIN {X 0,Y 117.264,Z 490.922,A -85,B 0,C 180,E1 -26770.679,E2 -26770.679} C_VEL
LIN {X 0,Y 120.928,Z 480.643,A -85,B 0,C 180,E1 -26773.073,E2 -26773.073} C_VEL
LIN {X 0,Y 124.059,Z 469.469,A -85,B 0,C 180,E1 -26775.087,E2 -26775.087} C_VEL
LIN {X 0,Y 126.799,Z 456.48,A -85,B 0,C 180,E1 -26776.758,E2 -26776.758} C_VEL
LIN {X 0,Y 128.835,Z 442.999,A -85,B 0,C 180,E1 -26777.856,E2 -26777.856} C_VEL
LIN {X 0,Y 130.131,Z 427.483,A -85,B 0,C 180,E1 -26778.599,E2 -26778.599} C_VEL
LIN {X 0,Y 130.119,Z 417.686,A -85,B 0,C 180,E1 -26779.336,E2 -26779.336} C_VEL
LIN {X 0,Y 129.526,Z 411.945,A -85,B 0,C 180,E1 -26780.017,E2 -26780.017} C_VEL
LIN {X 0,Y 128.185,Z 404.503,A -85,B 0,C 180,E1 -26781.17,E2 -26781.17} C_VEL
LIN {X 0,Y 126.336,Z 397.374,A -85,B 0,C 180,E1 -26782.575,E2 -26782.575} C_VEL
LIN {X 0,Y 123.015,Z 387.162,A -85,B 0,C 180,E1 -26785.079,E2 -26785.079} C_VEL
LIN {X 0,Y 120.794,Z 381.815,A -85,B 0,C 180,E1 -26786.77,E2 -26786.77} C_VEL
LIN {X 0,Y 115.362,Z 372.313,A -85,B 0,C 180,E1 -26791.112,E2 -26791.112} C_VEL
LIN {X 0,Y 112.188,Z 367.654,A -85,B 0,C 180,E1 -26793.99,E2 -26793.99} C_VEL
LIN {X 0,Y 109.917,Z 364.282,A -85,B 0,C 180,E1 -26796.313,E2 -26796.313} C_VEL
LIN {X 0,Y 107.425,Z 360.585,A -85,B 0,C 180,E1 -26799.192,E2 -26799.192} C_VEL
LIN {X 0,Y 104.47,Z 357.104,A -85,B 0,C 180,E1 -26803.048,E2 -26803.048} C_VEL
LIN {X 0,Y 103.457,Z 355.266,A -85,B 0,C 180,E1 -26804.672,E2 -26804.672} C_VEL
LIN {X 0,Y 101.187,Z 353.244,A -85,B 0,C 180,E1 -26808.48,E2 -26808.48} C_VEL
LIN {X 0,Y 99.669,Z 350.028,A -85,B 0,C 180,E1 -26812.158,E2 -26812.158} C_VEL
LIN {X 0,Y 99.363,Z 349.691,A -85,B 0,C 180,E1 -26812.934,E2 -26812.934} C_VEL
LIN {X 0,Y 97.373,Z 348.387,A -85,B 0,C 180,E1 -26819.482,E2 -26819.482} C_VEL
LIN {X 0,Y 96.553,Z 348.238,A -85,B 0,C 180,E1 -26828.37,E2 -26828.37} C_VEL
LIN {X 0,Y 99.341,Z 349.968,A -85,B 0,C 180,E1 -26841.562,E2 -26841.562} C_VEL
LIN {X 0,Y 100.364,Z 352.655,A -85,B 0,C 180,E1 -26844.392,E2 -26844.392} C_VEL
LIN {X 0,Y 102.887,Z 355.118,A -85,B 0,C 180,E1 -26848.989,E2 -26848.989} C_VEL
LIN {X 0,Y 103.701,Z 355.824,A -85,B 0,C 180,E1 -26850.225,E2 -26850.225} C_VEL
LIN {X 0,Y 105.684,Z 359.048,A -85,B 0,C 180,E1 -26853.168,E2 -26853.168} C_VEL
LIN {X 0,Y 107.52,Z 360.86,A -85,B 0,C 180,E1 -26855.405,E2 -26855.405} C_VEL
LIN {X 0,Y 110.162,Z 364.578,A -85,B 0,C 180,E1 -26858.402,E2 -26858.402} C_VEL
LIN {X 0,Y 113.965,Z 370.361,A -85,B 0,C 180,E1 -26862.142,E2 -26862.142} C_VEL
LIN {X 0,Y 117.682,Z 376.202,A -85,B 0,C 180,E1 -26865.293,E2 -26865.293} C_VEL
LIN {X 0,Y 122.063,Z 384.184,A -85,B 0,C 180,E1 -26868.616,E2 -26868.616} C_VEL
LIN {X 0,Y 126.709,Z 394.185,A -85,B 0,C 180,E1 -26871.808,E2 -26871.808} C_VEL
LIN {X 0,Y 127.327,Z 395.795,A -85,B 0,C 180,E1 -26872.224,E2 -26872.224} C_VEL
LIN {X 0,Y 123.706,Z 438.623,A -85,B 0,C 180,E1 -26874.169,E2 -26874.169} C_VEL
LIN {X 0,Y 121.61,Z 452.029,A -85,B 0,C 180,E1 -26875.324,E2 -26875.324} C_VEL
LIN {X 0,Y 118.716,Z 464.896,A -85,B 0,C 180,E1 -26877.047,E2 -26877.047} C_VEL
LIN {X 0,Y 115.387,Z 476.62,A -85,B 0,C 180,E1 -26879.326,E2 -26879.326} C_VEL
LIN {X 0,Y 111.406,Z 488.005,A -85,B 0,C 180,E1 -26882.29,E2 -26882.29} C_VEL
LIN {X 0,Y 107.172,Z 498.189,A -85,B 0,C 180,E1 -26885.801,E2 -26885.801} C_VEL
LIN {X 0,Y 103.026,Z 507.376,A -85,B 0,C 180,E1 -26890.054,E2 -26890.054} C_VEL
LIN {X 0,Y 98.716,Z 516.336,A -85,B 0,C 180,E1 -26895.567,E2 -26895.567} C_VEL
LIN {X 0,Y 95.342,Z 523.526,A -85,B 0,C 180,E1 -26901.518,E2 -26901.518} C_VEL
LIN {X 0,Y 92.921,Z 529.25,A -85,B 0,C 180,E1 -26907.829,E2 -26907.829} C_VEL
LIN {X 0,Y 91.431,Z 533.765,A -85,B 0,C 180,E1 -26914.404,E2 -26914.404} C_VEL
LIN {X 0,Y 90.74,Z 536.171,A -85,B 0,C 180,E1 -26918.907,E2 -26918.907} C_VEL
LIN {X 0,Y 90.481,Z 538.141,A -85,B 0,C 180,E1 -26923.471,E2 -26923.471} C_VEL
LIN {X 0,Y 90.721,Z 539.643,A -85,B 0,C 180,E1 -26928.047,E2 -26928.047} C_VEL
LIN {X 0,Y 91.391,Z 540.718,A -85,B 0,C 180,E1 -26932.663,E2 -26932.663} C_VEL
LIN {X 0,Y 92.415,Z 541.376,A -85,B 0,C 180,E1 -26937.143,E2 -26937.143} C_VEL
LIN {X 0,Y 93.987,Z 541.631,A -85,B 0,C 180,E1 -26941.558,E2 -26941.558} C_VEL
LIN {X 0,Y 96.696,Z 541.3,A -85,B 0,C 180,E1 -26946.919,E2 -26946.919} C_VEL
LIN {X 0,Y 101.525,Z 539.782,A -85,B 0,C 180,E1 -26953.803,E2 -26953.803} C_VEL
LIN {X 0,Y 105.928,Z 537.779,A -85,B 0,C 180,E1 -26958.436,E2 -26958.436} C_VEL
LIN {X 0,Y 112.856,Z 533.909,A -85,B 0,C 180,E1 -26964.047,E2 -26964.047} C_VEL
LIN {X 0,Y 119.756,Z 529.177,A -85,B 0,C 180,E1 -26968.481,E2 -26968.481} C_VEL
LIN {X 0,Y 127.001,Z 523.288,A -85,B 0,C 180,E1 -26972.295,E2 -26972.295} C_VEL
LIN {X 0,Y 135.3,Z 515.432,A -85,B 0,C 180,E1 -26975.783,E2 -26975.783} C_VEL
LIN {X 0,Y 143.325,Z 506.309,A -85,B 0,C 180,E1 -26978.689,E2 -26978.689} C_VEL
LIN {X 0,Y 150.561,Z 496.412,A -85,B 0,C 180,E1 -26980.929,E2 -26980.929} C_VEL
LIN {X 0,Y 157.237,Z 485.297,A -85,B 0,C 180,E1 -26982.813,E2 -26982.813} C_VEL
LIN {X 0,Y 162.542,Z 474.383,A -85,B 0,C 180,E1 -26984.154,E2 -26984.154} C_VEL
LIN {X 0,Y 167.135,Z 462.264,A -85,B 0,C 180,E1 -26985.262,E2 -26985.262} C_VEL
LIN {X 0,Y 170.505,Z 450.213,A -85,B 0,C 180,E1 -26986.076,E2 -26986.076} C_VEL
LIN {X 0,Y 172.997,Z 436.924,A -85,B 0,C 180,E1 -26986.641,E2 -26986.641} C_VEL
LIN {X 0,Y 173.34,Z 433.747,A -85,B 0,C 180,E1 -26986.78,E2 -26986.78} C_VEL
LIN {X 0,Y 170.822,Z 428.242,A -85,B 0,C 180,E1 -26989.942,E2 -26989.942} C_VEL
LIN {X 0,Y 168.499,Z 423.341,A -85,B 0,C 180,E1 -26993.565,E2 -26993.565} C_VEL
LIN {X 0,Y 166.858,Z 419.884,A -85,B 0,C 180,E1 -26996.983,E2 -26996.983} C_VEL
LIN {X 0,Y 165.56,Z 416.612,A -85,B 0,C 180,E1 -27001.217,E2 -27001.217} C_VEL
LIN {X 0,Y 164.818,Z 416.296,A -85,B 0,C 180,E1 -27008.23,E2 -27008.23} C_VEL
LIN {X 0,Y 165.514,Z 417.132,A -85,B 0,C 180,E1 -27012.507,E2 -27012.507} C_VEL
LIN {X 0,Y 167.015,Z 420.511,A -85,B 0,C 180,E1 -27017.132,E2 -27017.132} C_VEL
LIN {X 0,Y 168.548,Z 423.931,A -85,B 0,C 180,E1 -27020.281,E2 -27020.281} C_VEL
LIN {X 0,Y 170.604,Z 429.647,A -85,B 0,C 180,E1 -27023.682,E2 -27023.682} C_VEL
LIN {X 0,Y 173.075,Z 437.328,A -85,B 0,C 180,E1 -27027.072,E2 -27027.072} C_VEL
LIN {X 0,Y 171.104,Z 449.724,A -85,B 0,C 180,E1 -27027.557,E2 -27027.557} C_VEL
LIN {X 0,Y 168.168,Z 461.337,A -85,B 0,C 180,E1 -27028.176,E2 -27028.176} C_VEL
LIN {X 0,Y 163.778,Z 473.726,A -85,B 0,C 180,E1 -27029.04,E2 -27029.04} C_VEL
LIN {X 0,Y 158.575,Z 485.089,A -85,B 0,C 180,E1 -27030.21,E2 -27030.21} C_VEL
LIN {X 0,Y 152.018,Z 496.622,A -85,B 0,C 180,E1 -27031.848,E2 -27031.848} C_VEL
LIN {X 0,Y 145.619,Z 505.937,A -85,B 0,C 180,E1 -27033.645,E2 -27033.645} C_VEL
LIN {X 0,Y 138.74,Z 514.458,A -85,B 0,C 180,E1 -27035.861,E2 -27035.861} C_VEL
LIN {X 0,Y 130.823,Z 522.76,A -85,B 0,C 180,E1 -27038.839,E2 -27038.839} C_VEL
LIN {X 0,Y 123.266,Z 529.477,A -85,B 0,C 180,E1 -27042.172,E2 -27042.172} C_VEL
LIN {X 0,Y 116.311,Z 534.864,A -85,B 0,C 180,E1 -27045.987,E2 -27045.987} C_VEL
LIN {X 0,Y 110.081,Z 539.096,A -85,B 0,C 180,E1 -27050.329,E2 -27050.329} C_VEL
LIN {X 0,Y 106.269,Z 541.356,A -85,B 0,C 180,E1 -27053.477,E2 -27053.477} C_VEL
LIN {X 0,Y 102.752,Z 543.175,A -85,B 0,C 180,E1 -27056.831,E2 -27056.831} C_VEL
LIN {X 0,Y 96.967,Z 545.557,A -85,B 0,C 180,E1 -27064.227,E2 -27064.227} C_VEL
LIN {X 0,Y 93.149,Z 546.426,A -85,B 0,C 180,E1 -27072.439,E2 -27072.439} C_VEL
LIN {X 0,Y 91.989,Z 546.253,A -85,B 0,C 180,E1 -27076.754,E2 -27076.754} C_VEL
LIN {X 0,Y 91.004,Z 544.765,A -85,B 0,C 180,E1 -27085.575,E2 -27085.575} C_VEL
LIN {X 0,Y 91.05,Z 543.432,A -85,B 0,C 180,E1 -27090.004,E2 -27090.004} C_VEL
LIN {X 0,Y 91.063,Z 540.536,A -85,B 0,C 180,E1 -27096.652,E2 -27096.652} C_VEL
LIN {X 0,Y 91.852,Z 536.572,A -85,B 0,C 180,E1 -27103.274,E2 -27103.274} C_VEL
LIN {X 0,Y 93.969,Z 530.428,A -85,B 0,C 180,E1 -27110.813,E2 -27110.813} C_VEL
LIN {X 0,Y 97.069,Z 523.697,A -85,B 0,C 180,E1 -27116.909,E2 -27116.909} C_VEL
LIN {X 0,Y 100.976,Z 515.3,A -85,B 0,C 180,E1 -27122.647,E2 -27122.647} C_VEL
LIN {X 0,Y 104.426,Z 507.865,A -85,B 0,C 180,E1 -27126.499,E2 -27126.499} C_VEL
LIN {X 0,Y 108.619,Z 498.326,A -85,B 0,C 180,E1 -27130.322,E2 -27130.322} C_VEL
LIN {X 0,Y 111.98,Z 489.595,A -85,B 0,C 180,E1 -27133.046,E2 -27133.046} C_VEL
LIN {X 0,Y 115.784,Z 478.993,A -85,B 0,C 180,E1 -27135.501,E2 -27135.501} C_VEL
LIN {X 0,Y 119.114,Z 467.299,A -85,B 0,C 180,E1 -27137.525,E2 -27137.525} C_VEL
LIN {X 0,Y 121.889,Z 454.264,A -85,B 0,C 180,E1 -27139.134,E2 -27139.134} C_VEL
LIN {X 0,Y 123.789,Z 441.503,A -85,B 0,C 180,E1 -27140.113,E2 -27140.113} C_VEL
LIN {X 0,Y 126.925,Z 400.464,A -85,B 0,C 180,E1 -27142.054,E2 -27142.054} C_VEL
LIN {X 0,Y 126.442,Z 397.736,A -85,B 0,C 180,E1 -27142.496,E2 -27142.496} C_VEL
LIN {X 0,Y 126.336,Z 397.374,A -85,B 0,C 180,E1 -27142.575,E2 -27142.575} C_VEL
LIN {X 0,Y 124.356,Z 392.64,A -85,B 0,C 180,E1 -27143.923,E2 -27143.923} C_VEL
LIN {X 0,Y 120.825,Z 387.508,A -85,B 0,C 180,E1 -27146.231,E2 -27146.231} C_VEL
LIN {X 0,Y 112.324,Z 377.916,A -85,B 0,C 180,E1 -27152.696,E2 -27152.696} C_VEL
LIN {X 0,Y 107.725,Z 370.642,A -85,B 0,C 180,E1 -27157.489,E2 -27157.489} C_VEL
LIN {X 0,Y 104.607,Z 366.182,A -85,B 0,C 180,E1 -27161.405,E2 -27161.405} C_VEL
LIN {X 0,Y 102.233,Z 362.924,A -85,B 0,C 180,E1 -27164.93,E2 -27164.93} C_VEL
LIN {X 0,Y 101.553,Z 361.841,A -85,B 0,C 180,E1 -27166.105,E2 -27166.105} C_VEL
LIN {X 0,Y 99.192,Z 359.134,A -85,B 0,C 180,E1 -27170.697,E2 -27170.697} C_VEL
LIN {X 0,Y 98.058,Z 356.618,A -85,B 0,C 180,E1 -27173.918,E2 -27173.918} C_VEL
LIN {X 0,Y 96.379,Z 355.362,A -85,B 0,C 180,E1 -27179.999,E2 -27179.999} C_VEL
LIN {X 0,Y 95.785,Z 355.44,A -85,B 0,C 180,E1 -27190.528,E2 -27190.528} C_VEL
LIN {X 0,Y 97.98,Z 356.976,A -85,B 0,C 180,E1 -27200.467,E2 -27200.467} C_VEL
LIN {X 0,Y 99.326,Z 359.941,A -85,B 0,C 180,E1 -27204.233,E2 -27204.233} C_VEL
LIN {X 0,Y 101.838,Z 362.394,A -85,B 0,C 180,E1 -27208.886,E2 -27208.886} C_VEL
LIN {X 0,Y 104.076,Z 365.854,A -85,B 0,C 180,E1 -27212.397,E2 -27212.397} C_VEL
LIN {X 0,Y 105.51,Z 367.531,A -85,B 0,C 180,E1 -27214.272,E2 -27214.272} C_VEL
LIN {X 0,Y 108.397,Z 371.822,A -85,B 0,C 180,E1 -27217.757,E2 -27217.757} C_VEL
LIN {X 0,Y 112.632,Z 378.557,A -85,B 0,C 180,E1 -27222.071,E2 -27222.071} C_VEL
LIN {X 0,Y 117.301,Z 386.943,A -85,B 0,C 180,E1 -27226.117,E2 -27226.117} C_VEL
LIN {X 0,Y 122.156,Z 397.674,A -85,B 0,C 180,E1 -27229.857,E2 -27229.857} C_VEL
LIN {X 0,Y 120.431,Z 420.397,A -85,B 0,C 180,E1 -27230.948,E2 -27230.948} C_VEL
LIN {X 0,Y 118.526,Z 439.869,A -85,B 0,C 180,E1 -27231.892,E2 -27231.892} C_VEL
LIN {X 0,Y 116.432,Z 452.418,A -85,B 0,C 180,E1 -27233.003,E2 -27233.003} C_VEL
LIN {X 0,Y 113.385,Z 465.222,A -85,B 0,C 180,E1 -27234.741,E2 -27234.741} C_VEL
LIN {X 0,Y 109.877,Z 476.919,A -85,B 0,C 180,E1 -27237.062,E2 -27237.062} C_VEL
LIN {X 0,Y 105.692,Z 488.205,A -85,B 0,C 180,E1 -27240.068,E2 -27240.068} C_VEL
LIN {X 0,Y 101.189,Z 498.449,A -85,B 0,C 180,E1 -27243.715,E2 -27243.715} C_VEL
LIN {X 0,Y 96.339,Z 508.449,A -85,B 0,C 180,E1 -27248.604,E2 -27248.604} C_VEL
LIN {X 0,Y 91.822,Z 517.255,A -85,B 0,C 180,E1 -27254.457,E2 -27254.457} C_VEL
LIN {X 0,Y 88.308,Z 524.266,A -85,B 0,C 180,E1 -27260.837,E2 -27260.837} C_VEL
LIN {X 0,Y 85.775,Z 529.883,A -85,B 0,C 180,E1 -27267.648,E2 -27267.648} C_VEL
LIN {X 0,Y 84.217,Z 534.305,A -85,B 0,C 180,E1 -27274.783,E2 -27274.783} C_VEL
LIN {X 0,Y 83.552,Z 536.665,A -85,B 0,C 180,E1 -27279.68,E2 -27279.68} C_VEL
LIN {X 0,Y 83.388,Z 538.576,A -85,B 0,C 180,E1 -27284.641,E2 -27284.641} C_VEL
LIN {X 0,Y 84.429,Z 540.88,A -85,B 0,C 180,E1 -27293.703,E2 -27293.703} C_VEL
LIN {X 0,Y 85.899,Z 541.649,A -85,B 0,C 180,E1 -27299.395,E2 -27299.395} C_VEL
LIN {X 0,Y 87.747,Z 541.82,A -85,B 0,C 180,E1 -27304.096,E2 -27304.096} C_VEL
LIN {X 0,Y 90.331,Z 541.529,A -85,B 0,C 180,E1 -27308.921,E2 -27308.921} C_VEL
LIN {X 0,Y 96.282,Z 539.814,A -85,B 0,C 180,E1 -27316.875,E2 -27316.875} C_VEL
LIN {X 0,Y 100.431,Z 538.059,A -85,B 0,C 180,E1 -27320.966,E2 -27320.966} C_VEL
LIN {X 0,Y 106.372,Z 535.04,A -85,B 0,C 180,E1 -27325.671,E2 -27325.671} C_VEL
LIN {X 0,Y 113.847,Z 530.404,A -85,B 0,C 180,E1 -27330.407,E2 -27330.407} C_VEL
LIN {X 0,Y 122.381,Z 524.018,A -85,B 0,C 180,E1 -27334.745,E2 -27334.745} C_VEL
LIN {X 0,Y 129.858,Z 517.442,A -85,B 0,C 180,E1 -27337.739,E2 -27337.739} C_VEL
LIN {X 0,Y 137.862,Z 509.004,A -85,B 0,C 180,E1 -27340.57,E2 -27340.57} C_VEL
LIN {X 0,Y 145.299,Z 499.734,A -85,B 0,C 180,E1 -27342.793,E2 -27342.793} C_VEL
LIN {X 0,Y 152.13,Z 489.414,A -85,B 0,C 180,E1 -27344.647,E2 -27344.647} C_VEL
LIN {X 0,Y 158.348,Z 477.834,A -85,B 0,C 180,E1 -27346.128,E2 -27346.128} C_VEL
LIN {X 0,Y 163.313,Z 466.064,A -85,B 0,C 180,E1 -27347.27,E2 -27347.27} C_VEL
LIN {X 0,Y 167.182,Z 453.755,A -85,B 0,C 180,E1 -27348.157,E2 -27348.157} C_VEL
LIN {X 0,Y 170.07,Z 440.387,A -85,B 0,C 180,E1 -27348.757,E2 -27348.757} C_VEL
LIN {X 0,Y 170.435,Z 437.712,A -85,B 0,C 180,E1 -27348.927,E2 -27348.927} C_VEL
LIN {X 0,Y 168.223,Z 432.454,A -85,B 0,C 180,E1 -27352.348,E2 -27352.348} C_VEL
LIN {X 0,Y 166.856,Z 429.414,A -85,B 0,C 180,E1 -27354.865,E2 -27354.865} C_VEL
LIN {X 0,Y 165.705,Z 426.686,A -85,B 0,C 180,E1 -27357.57,E2 -27357.57} C_VEL
LIN {X 0,Y 164.522,Z 423.529,A -85,B 0,C 180,E1 -27361.837,E2 -27361.837} C_VEL
LIN {X 0,Y 163.941,Z 423.348,A -85,B 0,C 180,E1 -27368.274,E2 -27368.274} C_VEL
LIN {X 0,Y 164.528,Z 424.125,A -85,B 0,C 180,E1 -27372.123,E2 -27372.123} C_VEL
LIN {X 0,Y 166.256,Z 428.211,A -85,B 0,C 180,E1 -27377.53,E2 -27377.53} C_VEL
LIN {X 0,Y 167.413,Z 431.374,A -85,B 0,C 180,E1 -27380.024,E2 -27380.024} C_VEL
LIN {X 0,Y 168.981,Z 436.295,A -85,B 0,C 180,E1 -27382.869,E2 -27382.869} C_VEL
LIN {X 0,Y 170.245,Z 441.094,A -85,B 0,C 180,E1 -27385.004,E2 -27385.004} C_VEL
LIN {X 0,Y 167.628,Z 454.043,A -85,B 0,C 180,E1 -27385.5,E2 -27385.5} C_VEL
LIN {X 0,Y 163.601,Z 467.338,A -85,B 0,C 180,E1 -27386.271,E2 -27386.271} C_VEL
LIN {X 0,Y 158.939,Z 478.62,A -85,B 0,C 180,E1 -27387.147,E2 -27387.147} C_VEL
LIN {X 0,Y 152.889,Z 490.235,A -85,B 0,C 180,E1 -27388.467,E2 -27388.467} C_VEL
LIN {X 0,Y 146.227,Z 500.684,A -85,B 0,C 180,E1 -27390.109,E2 -27390.109} C_VEL
LIN {X 0,Y 138.947,Z 510.137,A -85,B 0,C 180,E1 -27392.095,E2 -27392.095} C_VEL
LIN {X 0,Y 130.557,Z 519.249,A -85,B 0,C 180,E1 -27394.829,E2 -27394.829} C_VEL
LIN {X 0,Y 122.513,Z 526.608,A -85,B 0,C 180,E1 -27397.935,E2 -27397.935} C_VEL
LIN {X 0,Y 113.653,Z 533.421,A -85,B 0,C 180,E1 -27402.099,E2 -27402.099} C_VEL
LIN {X 0,Y 106.632,Z 538.059,A -85,B 0,C 180,E1 -27406.47,E2 -27406.47} C_VEL
LIN {X 0,Y 100.655,Z 541.395,A -85,B 0,C 180,E1 -27411.073,E2 -27411.073} C_VEL
LIN {X 0,Y 96.869,Z 543.141,A -85,B 0,C 180,E1 -27414.525,E2 -27414.525} C_VEL
LIN {X 0,Y 90.618,Z 545.45,A -85,B 0,C 180,E1 -27422.273,E2 -27422.273} C_VEL
LIN {X 0,Y 88.204,Z 546.036,A -85,B 0,C 180,E1 -27426.527,E2 -27426.527} C_VEL
LIN {X 0,Y 85.066,Z 545.998,A -85,B 0,C 180,E1 -27435.654,E2 -27435.654} C_VEL
LIN {X 0,Y 83.915,Z 544.437,A -85,B 0,C 180,E1 -27445.2,E2 -27445.2} C_VEL
LIN {X 0,Y 83.948,Z 543.045,A -85,B 0,C 180,E1 -27450.004,E2 -27450.004} C_VEL
LIN {X 0,Y 83.996,Z 540.083,A -85,B 0,C 180,E1 -27457.214,E2 -27457.214} C_VEL
LIN {X 0,Y 84.932,Z 536.036,A -85,B 0,C 180,E1 -27464.378,E2 -27464.378} C_VEL
LIN {X 0,Y 87.334,Z 529.766,A -85,B 0,C 180,E1 -27472.477,E2 -27472.477} C_VEL
LIN {X 0,Y 90.75,Z 522.93,A -85,B 0,C 180,E1 -27478.953,E2 -27478.953} C_VEL
LIN {X 0,Y 94.282,Z 515.929,A -85,B 0,C 180,E1 -27483.996,E2 -27483.996} C_VEL
LIN {X 0,Y 97.547,Z 509.283,A -85,B 0,C 180,E1 -27487.765,E2 -27487.765} C_VEL
LIN {X 0,Y 102.258,Z 499.325,A -85,B 0,C 180,E1 -27492.079,E2 -27492.079} C_VEL
LIN {X 0,Y 106.322,Z 489.513,A -85,B 0,C 180,E1 -27495.287,E2 -27495.287} C_VEL
LIN {X 0,Y 110.314,Z 478.95,A -85,B 0,C 180,E1 -27497.788,E2 -27497.788} C_VEL
LIN {X 0,Y 113.808,Z 467.301,A -85,B 0,C 180,E1 -27499.84,E2 -27499.84} C_VEL
LIN {X 0,Y 116.769,Z 454.092,A -85,B 0,C 180,E1 -27501.489,E2 -27501.489} C_VEL
LIN {X 0,Y 118.788,Z 440.991,A -85,B 0,C 180,E1 -27502.49,E2 -27502.49} C_VEL
LIN {X 0,Y 121.964,Z 401.555,A -85,B 0,C 180,E1 -27504.371,E2 -27504.371} C_VEL
LIN {X 0,Y 118.893,Z 391.302,A -85,B 0,C 180,E1 -27506.977,E2 -27506.977} C_VEL
LIN {X 0,Y 116.853,Z 386.212,A -85,B 0,C 180,E1 -27508.699,E2 -27508.699} C_VEL
LIN {X 0,Y 112.324,Z 377.916,A -85,B 0,C 180,E1 -27512.696,E2 -27512.696} C_VEL
LIN {X 0,Y 109.809,Z 375.076,A -85,B 0,C 180,E1 -27515.048,E2 -27515.048} C_VEL
LIN {X 0,Y 105.531,Z 371.923,A -85,B 0,C 180,E1 -27519.506,E2 -27519.506} C_VEL
LIN {X 0,Y 99.695,Z 368.32,A -85,B 0,C 180,E1 -27527.65,E2 -27527.65} C_VEL
LIN {X 0,Y 97.528,Z 365.28,A -85,B 0,C 180,E1 -27532.528,E2 -27532.528} C_VEL
LIN {X 0,Y 96.911,Z 363.598,A -85,B 0,C 180,E1 -27534.572,E2 -27534.572} C_VEL
LIN {X 0,Y 95.482,Z 362.479,A -85,B 0,C 180,E1 -27539.999,E2 -27539.999} C_VEL
LIN {X 0,Y 94.799,Z 362.336,A -85,B 0,C 180,E1 -27548.526,E2 -27548.526} C_VEL
LIN {X 0,Y 96.703,Z 363.921,A -85,B 0,C 180,E1 -27559.437,E2 -27559.437} C_VEL
LIN {X 0,Y 97.993,Z 366.76,A -85,B 0,C 180,E1 -27563.351,E2 -27563.351} C_VEL
LIN {X 0,Y 100.134,Z 369.09,A -85,B 0,C 180,E1 -27567.679,E2 -27567.679} C_VEL
LIN {X 0,Y 102.469,Z 372.65,A -85,B 0,C 180,E1 -27571.577,E2 -27571.577} C_VEL
LIN {X 0,Y 103.64,Z 374.316,A -85,B 0,C 180,E1 -27573.247,E2 -27573.247} C_VEL
LIN {X 0,Y 106.197,Z 378.338,A -85,B 0,C 180,E1 -27576.555,E2 -27576.555} C_VEL
LIN {X 0,Y 109.565,Z 383.981,A -85,B 0,C 180,E1 -27580.306,E2 -27580.306} C_VEL
LIN {X 0,Y 113.739,Z 391.9,A -85,B 0,C 180,E1 -27584.313,E2 -27584.313} C_VEL
LIN {X 0,Y 117.352,Z 400.172,A -85,B 0,C 180,E1 -27587.427,E2 -27587.427} C_VEL
LIN {X 0,Y 114.08,Z 437.23,A -85,B 0,C 180,E1 -27589.147,E2 -27589.147} C_VEL
LIN {X 0,Y 111.843,Z 450.775,A -85,B 0,C 180,E1 -27590.236,E2 -27590.236} C_VEL
LIN {X 0,Y 108.856,Z 463.418,A -85,B 0,C 180,E1 -27591.871,E2 -27591.871} C_VEL
LIN {X 0,Y 105.105,Z 475.639,A -85,B 0,C 180,E1 -27594.187,E2 -27594.187} C_VEL
LIN {X 0,Y 100.994,Z 486.464,A -85,B 0,C 180,E1 -27597.016,E2 -27597.016} C_VEL
LIN {X 0,Y 95.865,Z 497.677,A -85,B 0,C 180,E1 -27600.938,E2 -27600.938} C_VEL
LIN {X 0,Y 91.543,Z 506.21,A -85,B 0,C 180,E1 -27605.019,E2 -27605.019} C_VEL
LIN {X 0,Y 86.443,Z 515.453,A -85,B 0,C 180,E1 -27611.018,E2 -27611.018} C_VEL
LIN {X 0,Y 82.363,Z 522.881,A -85,B 0,C 180,E1 -27617.678,E2 -27617.678} C_VEL
LIN {X 0,Y 79.347,Z 528.84,A -85,B 0,C 180,E1 -27624.914,E2 -27624.914} C_VEL
LIN {X 0,Y 77.407,Z 533.717,A -85,B 0,C 180,E1 -27632.915,E2 -27632.915} C_VEL
LIN {X 0,Y 76.373,Z 537.161,A -85,B 0,C 180,E1 -27640.6,E2 -27640.6} C_VEL
LIN {X 0,Y 76.328,Z 538.982,A -85,B 0,C 180,E1 -27646.03,E2 -27646.03} C_VEL
LIN {X 0,Y 77.543,Z 541.054,A -85,B 0,C 180,E1 -27655,E2 -27655} C_VEL
LIN {X 0,Y 79.521,Z 541.9,A -85,B 0,C 180,E1 -27662.018,E2 -27662.018} C_VEL
LIN {X 0,Y 84.096,Z 541.757,A -85,B 0,C 180,E1 -27671.226,E2 -27671.226} C_VEL
LIN {X 0,Y 87.663,Z 540.998,A -85,B 0,C 180,E1 -27676.175,E2 -27676.175} C_VEL
LIN {X 0,Y 91.345,Z 539.819,A -85,B 0,C 180,E1 -27680.293,E2 -27680.293} C_VEL
LIN {X 0,Y 97.704,Z 537.231,A -85,B 0,C 180,E1 -27685.806,E2 -27685.806} C_VEL
LIN {X 0,Y 104.811,Z 533.557,A -85,B 0,C 180,E1 -27690.649,E2 -27690.649} C_VEL
LIN {X 0,Y 112.558,Z 528.683,A -85,B 0,C 180,E1 -27694.864,E2 -27694.864} C_VEL
LIN {X 0,Y 120.846,Z 522.46,A -85,B 0,C 180,E1 -27698.505,E2 -27698.505} C_VEL
LIN {X 0,Y 129.577,Z 514.657,A -85,B 0,C 180,E1 -27701.642,E2 -27701.642} C_VEL
LIN {X 0,Y 137.115,Z 506.582,A -85,B 0,C 180,E1 -27703.946,E2 -27703.946} C_VEL
LIN {X 0,Y 144.85,Z 496.645,A -85,B 0,C 180,E1 -27706.009,E2 -27706.009} C_VEL
LIN {X 0,Y 151.145,Z 486.854,A -85,B 0,C 180,E1 -27707.533,E2 -27707.533} C_VEL
LIN {X 0,Y 156.742,Z 476.285,A -85,B 0,C 180,E1 -27708.749,E2 -27708.749} C_VEL
LIN {X 0,Y 161.57,Z 464.724,A -85,B 0,C 180,E1 -27709.75,E2 -27709.75} C_VEL
LIN {X 0,Y 165.616,Z 451.437,A -85,B 0,C 180,E1 -27710.598,E2 -27710.598} C_VEL
LIN {X 0,Y 167.676,Z 441.967,A -85,B 0,C 180,E1 -27711.001,E2 -27711.001} C_VEL
LIN {X 0,Y 165.851,Z 436.774,A -85,B 0,C 180,E1 -27714.834,E2 -27714.834} C_VEL
LIN {X 0,Y 164.571,Z 433.46,A -85,B 0,C 180,E1 -27718.165,E2 -27718.165} C_VEL
LIN {X 0,Y 163.506,Z 430.427,A -85,B 0,C 180,E1 -27722.464,E2 -27722.464} C_VEL
LIN {X 0,Y 163.13,Z 430.468,A -85,B 0,C 180,E1 -27729.045,E2 -27729.045} C_VEL
LIN {X 0,Y 163.528,Z 431.064,A -85,B 0,C 180,E1 -27731.623,E2 -27731.623} C_VEL
LIN {X 0,Y 164.985,Z 434.785,A -85,B 0,C 180,E1 -27736.711,E2 -27736.711} C_VEL
LIN {X 0,Y 165.94,Z 437.875,A -85,B 0,C 180,E1 -27739.162,E2 -27739.162} C_VEL
LIN {X 0,Y 167.205,Z 443.089,A -85,B 0,C 180,E1 -27742.147,E2 -27742.147} C_VEL
LIN {X 0,Y 167.481,Z 444.375,A -85,B 0,C 180,E1 -27742.775,E2 -27742.775} C_VEL
LIN {X 0,Y 164.512,Z 457.412,A -85,B 0,C 180,E1 -27743.343,E2 -27743.343} C_VEL
LIN {X 0,Y 160.607,Z 469.045,A -85,B 0,C 180,E1 -27744.018,E2 -27744.018} C_VEL
LIN {X 0,Y 155.073,Z 481.431,A -85,B 0,C 180,E1 -27744.993,E2 -27744.993} C_VEL
LIN {X 0,Y 148.885,Z 492.49,A -85,B 0,C 180,E1 -27746.256,E2 -27746.256} C_VEL
LIN {X 0,Y 142.816,Z 501.456,A -85,B 0,C 180,E1 -27747.658,E2 -27747.658} C_VEL
LIN {X 0,Y 135.329,Z 510.697,A -85,B 0,C 180,E1 -27749.562,E2 -27749.562} C_VEL
LIN {X 0,Y 126.647,Z 519.667,A -85,B 0,C 180,E1 -27752.199,E2 -27752.199} C_VEL
LIN {X 0,Y 118.286,Z 526.918,A -85,B 0,C 180,E1 -27755.224,E2 -27755.224} C_VEL
LIN {X 0,Y 111.59,Z 531.849,A -85,B 0,C 180,E1 -27758.076,E2 -27758.076} C_VEL
LIN {X 0,Y 104.13,Z 536.656,A -85,B 0,C 180,E1 -27762.068,E2 -27762.068} C_VEL
LIN {X 0,Y 97.358,Z 540.373,A -85,B 0,C 180,E1 -27766.709,E2 -27766.709} C_VEL
LIN {X 0,Y 91.168,Z 543.108,A -85,B 0,C 180,E1 -27771.929,E2 -27771.929} C_VEL
LIN {X 0,Y 84.395,Z 545.343,A -85,B 0,C 180,E1 -27780.028,E2 -27780.028} C_VEL
LIN {X 0,Y 81.711,Z 545.871,A -85,B 0,C 180,E1 -27784.534,E2 -27784.534} C_VEL
LIN {X 0,Y 78.189,Z 545.744,A -85,B 0,C 180,E1 -27794.361,E2 -27794.361} C_VEL
LIN {X 0,Y 76.851,Z 544.106,A -85,B 0,C 180,E1 -27804.758,E2 -27804.758} C_VEL
LIN {X 0,Y 76.855,Z 542.642,A -85,B 0,C 180,E1 -27810.005,E2 -27810.005} C_VEL
LIN {X 0,Y 76.954,Z 539.604,A -85,B 0,C 180,E1 -27817.878,E2 -27817.878} C_VEL
LIN {X 0,Y 78.029,Z 535.468,A -85,B 0,C 180,E1 -27825.681,E2 -27825.681} C_VEL
LIN {X 0,Y 80.786,Z 529.103,A -85,B 0,C 180,E1 -27834.413,E2 -27834.413} C_VEL
LIN {X 0,Y 84.543,Z 522.161,A -85,B 0,C 180,E1 -27841.307,E2 -27841.307} C_VEL
LIN {X 0,Y 88.194,Z 515.385,A -85,B 0,C 180,E1 -27846.379,E2 -27846.379} C_VEL
LIN {X 0,Y 92.987,Z 506.433,A -85,B 0,C 180,E1 -27851.405,E2 -27851.405} C_VEL
LIN {X 0,Y 98.097,Z 495.755,A -85,B 0,C 180,E1 -27855.766,E2 -27855.766} C_VEL
LIN {X 0,Y 101.464,Z 488.063,A -85,B 0,C 180,E1 -27858.13,E2 -27858.13} C_VEL
LIN {X 0,Y 105.598,Z 477.109,A -85,B 0,C 180,E1 -27860.692,E2 -27860.692} C_VEL
LIN {X 0,Y 109.292,Z 465.004,A -85,B 0,C 180,E1 -27862.733,E2 -27862.733} C_VEL
LIN {X 0,Y 112.141,Z 452.608,A -85,B 0,C 180,E1 -27864.18,E2 -27864.18} C_VEL
LIN {X 0,Y 114.071,Z 440.078,A -85,B 0,C 180,E1 -27865.081,E2 -27865.081} C_VEL
LIN {X 0,Y 117.15,Z 403.288,A -85,B 0,C 180,E1 -27866.859,E2 -27866.859} C_VEL
LIN {X 0,Y 114.199,Z 393.314,A -85,B 0,C 180,E1 -27869.693,E2 -27869.693} C_VEL
LIN {X 0,Y 111.602,Z 387.79,A -85,B 0,C 180,E1 -27872.12,E2 -27872.12} C_VEL
LIN {X 0,Y 107.682,Z 380.585,A -85,B 0,C 180,E1 -27876.204,E2 -27876.204} C_VEL
LIN {X 0,Y 104.75,Z 375.973,A -85,B 0,C 180,E1 -27879.735,E2 -27879.735} C_VEL
LIN {X 0,Y 102.517,Z 372.452,A -85,B 0,C 180,E1 -27882.867,E2 -27882.867} C_VEL
LIN {X 0,Y 100.201,Z 368.959,A -85,B 0,C 180,E1 -27886.712,E2 -27886.712} C_VEL
LIN {X 0,Y 99.695,Z 368.32,A -85,B 0,C 180,E1 -27887.65,E2 -27887.65} C_VEL
LIN {X 0,Y 98.012,Z 367.405,A -85,B 0,C 180,E1 -27890.91,E2 -27890.91} C_VEL
LIN {X 0,Y 95.682,Z 367.765,A -85,B 0,C 180,E1 -27896.633,E2 -27896.633} C_VEL
LIN {X 0,Y 94.075,Z 369.146,A -85,B 0,C 180,E1 -27903.851,E2 -27903.851} C_VEL
LIN {X 0,Y 93.907,Z 369.338,A -85,B 0,C 180,E1 -27906.307,E2 -27906.307} C_VEL
LIN {X 0,Y 94.669,Z 370.178,A -85,B 0,C 180,E1 -27915.17,E2 -27915.17} C_VEL
LIN {X 0,Y 95.461,Z 370.851,A -85,B 0,C 180,E1 -27918.381,E2 -27918.381} C_VEL
LIN {X 0,Y 97.01,Z 374.013,A -85,B 0,C 180,E1 -27923.262,E2 -27923.262} C_VEL
LIN {X 0,Y 98.505,Z 375.796,A -85,B 0,C 180,E1 -27926.483,E2 -27926.483} C_VEL
LIN {X 0,Y 101.518,Z 380.547,A -85,B 0,C 180,E1 -27931.738,E2 -27931.738} C_VEL
LIN {X 0,Y 104.346,Z 385.267,A -85,B 0,C 180,E1 -27935.676,E2 -27935.676} C_VEL
LIN {X 0,Y 108.154,Z 392.403,A -85,B 0,C 180,E1 -27940.167,E2 -27940.167} C_VEL
LIN {X 0,Y 111.288,Z 399.183,A -85,B 0,C 180,E1 -27943.384,E2 -27943.384} C_VEL
LIN {X 0,Y 112.803,Z 403.084,A -85,B 0,C 180,E1 -27944.857,E2 -27944.857} C_VEL
LIN {X 0,Y 109.289,Z 438.808,A -85,B 0,C 180,E1 -27946.445,E2 -27946.445} C_VEL
LIN {X 0,Y 106.873,Z 452.497,A -85,B 0,C 180,E1 -27947.627,E2 -27947.627} C_VEL
LIN {X 0,Y 103.672,Z 464.868,A -85,B 0,C 180,E1 -27949.267,E2 -27949.267} C_VEL
LIN {X 0,Y 100.036,Z 475.938,A -85,B 0,C 180,E1 -27951.423,E2 -27951.423} C_VEL
LIN {X 0,Y 95.41,Z 487.323,A -85,B 0,C 180,E1 -27954.451,E2 -27954.451} C_VEL
LIN {X 0,Y 90.246,Z 497.943,A -85,B 0,C 180,E1 -27958.283,E2 -27958.283} C_VEL
LIN {X 0,Y 85.153,Z 507.303,A -85,B 0,C 180,E1 -27962.999,E2 -27962.999} C_VEL
LIN {X 0,Y 79.726,Z 516.379,A -85,B 0,C 180,E1 -27969.349,E2 -27969.349} C_VEL
LIN {X 0,Y 75.387,Z 523.681,A -85,B 0,C 180,E1 -27976.518,E2 -27976.518} C_VEL
LIN {X 0,Y 72.213,Z 529.513,A -85,B 0,C 180,E1 -27984.41,E2 -27984.41} C_VEL
LIN {X 0,Y 70.341,Z 533.899,A -85,B 0,C 180,E1 -27992.41,E2 -27992.41} C_VEL
LIN {X 0,Y 69.22,Z 537.633,A -85,B 0,C 180,E1 -28001.711,E2 -28001.711} C_VEL
LIN {X 0,Y 69.331,Z 539.385,A -85,B 0,C 180,E1 -28007.699,E2 -28007.699} C_VEL
LIN {X 0,Y 70.671,Z 541.219,A -85,B 0,C 180,E1 -28016.491,E2 -28016.491} C_VEL
LIN {X 0,Y 73.328,Z 542.13,A -85,B 0,C 180,E1 -28025.097,E2 -28025.097} C_VEL
LIN {X 0,Y 78.033,Z 541.984,A -85,B 0,C 180,E1 -28033.905,E2 -28033.905} C_VEL
LIN {X 0,Y 82.673,Z 541.064,A -85,B 0,C 180,E1 -28039.907,E2 -28039.907} C_VEL
LIN {X 0,Y 90.144,Z 538.615,A -85,B 0,C 180,E1 -28046.925,E2 -28046.925} C_VEL
LIN {X 0,Y 98.742,Z 534.761,A -85,B 0,C 180,E1 -28052.826,E2 -28052.826} C_VEL
LIN {X 0,Y 106.8,Z 530.205,A -85,B 0,C 180,E1 -28057.103,E2 -28057.103} C_VEL
LIN {X 0,Y 115.366,Z 524.341,A -85,B 0,C 180,E1 -28060.767,E2 -28060.767} C_VEL
LIN {X 0,Y 124.378,Z 516.91,A -85,B 0,C 180,E1 -28063.848,E2 -28063.848} C_VEL
LIN {X 0,Y 132.104,Z 509.287,A -85,B 0,C 180,E1 -28066.132,E2 -28066.132} C_VEL
LIN {X 0,Y 140.216,Z 499.783,A -85,B 0,C 180,E1 -28068.162,E2 -28068.162} C_VEL
LIN {X 0,Y 147.284,Z 489.661,A -85,B 0,C 180,E1 -28069.776,E2 -28069.776} C_VEL
LIN {X 0,Y 153.834,Z 478.067,A -85,B 0,C 180,E1 -28071.079,E2 -28071.079} C_VEL
LIN {X 0,Y 159.169,Z 465.991,A -85,B 0,C 180,E1 -28072.108,E2 -28072.108} C_VEL
LIN {X 0,Y 163.369,Z 452.968,A -85,B 0,C 180,E1 -28072.919,E2 -28072.919} C_VEL
LIN {X 0,Y 164.984,Z 446.337,A -85,B 0,C 180,E1 -28073.211,E2 -28073.211} C_VEL
LIN {X 0,Y 163.967,Z 442.809,A -85,B 0,C 180,E1 -28076.16,E2 -28076.16} C_VEL
LIN {X 0,Y 163.115,Z 439.916,A -85,B 0,C 180,E1 -28079.229,E2 -28079.229} C_VEL
LIN {X 0,Y 162.533,Z 437.488,A -85,B 0,C 180,E1 -28082.479,E2 -28082.479} C_VEL
LIN {X 0,Y 162.148,Z 437.468,A -85,B 0,C 180,E1 -28088.726,E2 -28088.726} C_VEL
LIN {X 0,Y 162.481,Z 438.022,A -85,B 0,C 180,E1 -28091.225,E2 -28091.225} C_VEL
LIN {X 0,Y 163.641,Z 441.669,A -85,B 0,C 180,E1 -28096.211,E2 -28096.211} C_VEL
LIN {X 0,Y 164.299,Z 444.582,A -85,B 0,C 180,E1 -28098.471,E2 -28098.471} C_VEL
LIN {X 0,Y 164.873,Z 447.986,A -85,B 0,C 180,E1 -28100.499,E2 -28100.499} C_VEL
LIN {X 0,Y 162.362,Z 458.04,A -85,B 0,C 180,E1 -28100.979,E2 -28100.979} C_VEL
LIN {X 0,Y 157.872,Z 470.696,A -85,B 0,C 180,E1 -28101.682,E2 -28101.682} C_VEL
LIN {X 0,Y 152.235,Z 482.694,A -85,B 0,C 180,E1 -28102.592,E2 -28102.592} C_VEL
LIN {X 0,Y 145.905,Z 493.403,A -85,B 0,C 180,E1 -28103.773,E2 -28103.773} C_VEL
LIN {X 0,Y 138.145,Z 504.113,A -85,B 0,C 180,E1 -28105.45,E2 -28105.45} C_VEL
LIN {X 0,Y 131.988,Z 511.237,A -85,B 0,C 180,E1 -28106.895,E2 -28106.895} C_VEL
LIN {X 0,Y 123.023,Z 520.084,A -85,B 0,C 180,E1 -28109.409,E2 -28109.409} C_VEL
LIN {X 0,Y 114.35,Z 527.225,A -85,B 0,C 180,E1 -28112.326,E2 -28112.326} C_VEL
LIN {X 0,Y 107.359,Z 532.063,A -85,B 0,C 180,E1 -28115.093,E2 -28115.093} C_VEL
LIN {X 0,Y 99.512,Z 536.782,A -85,B 0,C 180,E1 -28119.031,E2 -28119.031} C_VEL
LIN {X 0,Y 92.294,Z 540.418,A -85,B 0,C 180,E1 -28123.67,E2 -28123.67} C_VEL
LIN {X 0,Y 85.681,Z 543.074,A -85,B 0,C 180,E1 -28128.995,E2 -28128.995} C_VEL
LIN {X 0,Y 78.324,Z 545.228,A -85,B 0,C 180,E1 -28137.432,E2 -28137.432} C_VEL
LIN {X 0,Y 75.337,Z 545.69,A -85,B 0,C 180,E1 -28142.202,E2 -28142.202} C_VEL
LIN {X 0,Y 71.369,Z 545.49,A -85,B 0,C 180,E1 -28152.823,E2 -28152.823} C_VEL
LIN {X 0,Y 70.252,Z 544.827,A -85,B 0,C 180,E1 -28158.464,E2 -28158.464} C_VEL
LIN {X 0,Y 69.776,Z 543.75,A -85,B 0,C 180,E1 -28164.225,E2 -28164.225} C_VEL
LIN {X 0,Y 69.752,Z 542.239,A -85,B 0,C 180,E1 -28170.005,E2 -28170.005} C_VEL
LIN {X 0,Y 69.918,Z 539.121,A -85,B 0,C 180,E1 -28178.677,E2 -28178.677} C_VEL
LIN {X 0,Y 71.185,Z 534.898,A -85,B 0,C 180,E1 -28187.234,E2 -28187.234} C_VEL
LIN {X 0,Y 74.352,Z 528.442,A -85,B 0,C 180,E1 -28196.684,E2 -28196.684} C_VEL
LIN {X 0,Y 78.484,Z 521.369,A -85,B 0,C 180,E1 -28204.038,E2 -28204.038} C_VEL
LIN {X 0,Y 82.338,Z 514.716,A -85,B 0,C 180,E1 -28209.206,E2 -28209.206} C_VEL
LIN {X 0,Y 87.731,Z 505.329,A -85,B 0,C 180,E1 -28214.509,E2 -28214.509} C_VEL
LIN {X 0,Y 92.667,Z 495.663,A -85,B 0,C 180,E1 -28218.503,E2 -28218.503} C_VEL
LIN {X 0,Y 96.228,Z 487.993,A -85,B 0,C 180,E1 -28220.901,E2 -28220.901} C_VEL
LIN {X 0,Y 100.579,Z 477.068,A -85,B 0,C 180,E1 -28223.477,E2 -28223.477} C_VEL
LIN {X 0,Y 104.456,Z 465.006,A -85,B 0,C 180,E1 -28225.513,E2 -28225.513} C_VEL
LIN {X 0,Y 107.598,Z 451.828,A -85,B 0,C 180,E1 -28227.032,E2 -28227.032} C_VEL
LIN {X 0,Y 109.649,Z 438.581,A -85,B 0,C 180,E1 -28227.934,E2 -28227.934} C_VEL
LIN {X 0,Y 112.566,Z 405.23,A -85,B 0,C 180,E1 -28229.541,E2 -28229.541} C_VEL
LIN {X 0,Y 110.059,Z 396.481,A -85,B 0,C 180,E1 -28232.292,E2 -28232.292} C_VEL
LIN {X 0,Y 106.133,Z 388.411,A -85,B 0,C 180,E1 -28236.589,E2 -28236.589} C_VEL
LIN {X 0,Y 102.53,Z 382.121,A -85,B 0,C 180,E1 -28241.257,E2 -28241.257} C_VEL
LIN {X 0,Y 100.452,Z 378.711,A -85,B 0,C 180,E1 -28244.452,E2 -28244.452} C_VEL
LIN {X 0,Y 98.061,Z 374.906,A -85,B 0,C 180,E1 -28248.959,E2 -28248.959} C_VEL
LIN {X 0,Y 95.982,Z 371.498,A -85,B 0,C 180,E1 -28254.359,E2 -28254.359} C_VEL
LIN {X 0,Y 95.61,Z 370.448,A -85,B 0,C 180,E1 -28255.784,E2 -28255.784} C_VEL
LIN {X 0,Y 94.245,Z 369.384,A -85,B 0,C 180,E1 -28262.136,E2 -28262.136} C_VEL
LIN {X 0,Y 93.907,Z 369.338,A -85,B 0,C 180,E1 -28266.307,E2 -28266.307} C_VEL
LIN {X 0,Y 93.851,Z 369.983,A -85,B 0,C 180,E1 -28268.674,E2 -28268.674} C_VEL
LIN {X 0,Y 93.817,Z 371.502,A -85,B 0,C 180,E1 -28270.917,E2 -28270.917} C_VEL
LIN {X 0,Y 94.428,Z 378.267,A -85,B 0,C 180,E1 -28278.09,E2 -28278.09} C_VEL
LIN {X 0,Y 96.4,Z 381.665,A -85,B 0,C 180,E1 -28284.043,E2 -28284.043} C_VEL
LIN {X 0,Y 99.456,Z 386.698,A -85,B 0,C 180,E1 -28290.132,E2 -28290.132} C_VEL
LIN {X 0,Y 102.419,Z 392.12,A -85,B 0,C 180,E1 -28294.651,E2 -28294.651} C_VEL
LIN {X 0,Y 106.062,Z 399.662,A -85,B 0,C 180,E1 -28299.288,E2 -28299.288} C_VEL
LIN {X 0,Y 108.337,Z 405.31,A -85,B 0,C 180,E1 -28301.87,E2 -28301.87} C_VEL
LIN {X 0,Y 107.053,Z 419.964,A -85,B 0,C 180,E1 -28302.592,E2 -28302.592} C_VEL
LIN {X 0,Y 104.837,Z 440.179,A -85,B 0,C 180,E1 -28303.53,E2 -28303.53} C_VEL
LIN {X 0,Y 102.382,Z 453.097,A -85,B 0,C 180,E1 -28304.644,E2 -28304.644} C_VEL
LIN {X 0,Y 99.056,Z 465.2,A -85,B 0,C 180,E1 -28306.226,E2 -28306.226} C_VEL
LIN {X 0,Y 94.609,Z 477.816,A -85,B 0,C 180,E1 -28308.75,E2 -28308.75} C_VEL
LIN {X 0,Y 89.86,Z 488.557,A -85,B 0,C 180,E1 -28311.688,E2 -28311.688} C_VEL
LIN {X 0,Y 84.268,Z 499.229,A -85,B 0,C 180,E1 -28315.735,E2 -28315.735} C_VEL
LIN {X 0,Y 78.86,Z 508.375,A -85,B 0,C 180,E1 -28320.644,E2 -28320.644} C_VEL
LIN {X 0,Y 73.101,Z 517.303,A -85,B 0,C 180,E1 -28327.378,E2 -28327.378} C_VEL
LIN {X 0,Y 68.473,Z 524.451,A -85,B 0,C 180,E1 -28335.126,E2 -28335.126} C_VEL
LIN {X 0,Y 65.093,Z 530.149,A -85,B 0,C 180,E1 -28343.796,E2 -28343.796} C_VEL
LIN {X 0,Y 63.279,Z 534.046,A -85,B 0,C 180,E1 -28351.709,E2 -28351.709} C_VEL
LIN {X 0,Y 62.09,Z 538.081,A -85,B 0,C 180,E1 -28363.078,E2 -28363.078} C_VEL
LIN {X 0,Y 62.385,Z 539.79,A -85,B 0,C 180,E1 -28369.747,E2 -28369.747} C_VEL
LIN {X 0,Y 63.838,Z 541.38,A -85,B 0,C 180,E1 -28378.273,E2 -28378.273} C_VEL
LIN {X 0,Y 67.381,Z 542.36,A -85,B 0,C 180,E1 -28388.734,E2 -28388.734} C_VEL
LIN {X 0,Y 72.22,Z 542.206,A -85,B 0,C 180,E1 -28397.065,E2 -28397.065} C_VEL
LIN {X 0,Y 78.089,Z 541.115,A -85,B 0,C 180,E1 -28404.087,E2 -28404.087} C_VEL
LIN {X 0,Y 85.45,Z 538.887,A -85,B 0,C 180,E1 -28410.432,E2 -28410.432} C_VEL
LIN {X 0,Y 92.846,Z 535.892,A -85,B 0,C 180,E1 -28415.267,E2 -28415.267} C_VEL
LIN {X 0,Y 101.643,Z 531.383,A -85,B 0,C 180,E1 -28419.775,E2 -28419.775} C_VEL
LIN {X 0,Y 111.61,Z 525.051,A -85,B 0,C 180,E1 -28423.785,E2 -28423.785} C_VEL
LIN {X 0,Y 120.888,Z 517.838,A -85,B 0,C 180,E1 -28426.698,E2 -28426.698} C_VEL
LIN {X 0,Y 128.92,Z 510.311,A -85,B 0,C 180,E1 -28428.872,E2 -28428.872} C_VEL
LIN {X 0,Y 137.575,Z 500.576,A -85,B 0,C 180,E1 -28430.85,E2 -28430.85} C_VEL
LIN {X 0,Y 144.493,Z 491.103,A -85,B 0,C 180,E1 -28432.294,E2 -28432.294} C_VEL
LIN {X 0,Y 151.186,Z 479.875,A -85,B 0,C 180,E1 -28433.507,E2 -28433.507} C_VEL
LIN {X 0,Y 156.693,Z 468.068,A -85,B 0,C 180,E1 -28434.478,E2 -28434.478} C_VEL
LIN {X 0,Y 161.201,Z 455.207,A -85,B 0,C 180,E1 -28435.268,E2 -28435.268} C_VEL
LIN {X 0,Y 162.381,Z 450.854,A -85,B 0,C 180,E1 -28435.468,E2 -28435.468} C_VEL
LIN {X 0,Y 161.509,Z 446.709,A -85,B 0,C 180,E1 -28439.689,E2 -28439.689} C_VEL
LIN {X 0,Y 161.136,Z 444.416,A -85,B 0,C 180,E1 -28443.087,E2 -28443.087} C_VEL
LIN {X 0,Y 160.898,Z 444.457,A -85,B 0,C 180,E1 -28448.794,E2 -28448.794} C_VEL
LIN {X 0,Y 161.133,Z 444.944,A -85,B 0,C 180,E1 -28450.842,E2 -28450.842} C_VEL
LIN {X 0,Y 161.951,Z 448.468,A -85,B 0,C 180,E1 -28455.738,E2 -28455.738} C_VEL
LIN {X 0,Y 162.397,Z 451.965,A -85,B 0,C 180,E1 -28458.257,E2 -28458.257} C_VEL
LIN {X 0,Y 158.76,Z 463.925,A -85,B 0,C 180,E1 -28458.808,E2 -28458.808} C_VEL
LIN {X 0,Y 153.759,Z 475.954,A -85,B 0,C 180,E1 -28459.494,E2 -28459.494} C_VEL
LIN {X 0,Y 148.07,Z 486.721,A -85,B 0,C 180,E1 -28460.386,E2 -28460.386} C_VEL
LIN {X 0,Y 140.821,Z 497.749,A -85,B 0,C 180,E1 -28461.647,E2 -28461.647} C_VEL
LIN {X 0,Y 132.069,Z 508.471,A -85,B 0,C 180,E1 -28463.38,E2 -28463.38} C_VEL
LIN {X 0,Y 124.315,Z 516.398,A -85,B 0,C 180,E1 -28465.247,E2 -28465.247} C_VEL
LIN {X 0,Y 115.175,Z 524.207,A -85,B 0,C 180,E1 -28467.782,E2 -28467.782} C_VEL
LIN {X 0,Y 106.326,Z 530.471,A -85,B 0,C 180,E1 -28470.771,E2 -28470.771} C_VEL
LIN {X 0,Y 97.88,Z 535.482,A -85,B 0,C 180,E1 -28474.345,E2 -28474.345} C_VEL
LIN {X 0,Y 88.54,Z 540.021,A -85,B 0,C 180,E1 -28479.616,E2 -28479.616} C_VEL
LIN {X 0,Y 80.451,Z 543.041,A -85,B 0,C 180,E1 -28485.671,E2 -28485.671} C_VEL
LIN {X 0,Y 76.22,Z 544.275,A -85,B 0,C 180,E1 -28489.807,E2 -28489.807} C_VEL
LIN {X 0,Y 69.112,Z 545.508,A -85,B 0,C 180,E1 -28499.446,E2 -28499.446} C_VEL
LIN {X 0,Y 64.589,Z 545.236,A -85,B 0,C 180,E1 -28510.954,E2 -28510.954} C_VEL
LIN {X 0,Y 63.3,Z 544.525,A -85,B 0,C 180,E1 -28517.176,E2 -28517.176} C_VEL
LIN {X 0,Y 62.727,Z 543.386,A -85,B 0,C 180,E1 -28523.573,E2 -28523.573} C_VEL
LIN {X 0,Y 62.673,Z 541.837,A -85,B 0,C 180,E1 -28530.006,E2 -28530.006} C_VEL
LIN {X 0,Y 62.883,Z 538.636,A -85,B 0,C 180,E1 -28539.657,E2 -28539.657} C_VEL
LIN {X 0,Y 64.414,Z 534.329,A -85,B 0,C 180,E1 -28549.112,E2 -28549.112} C_VEL
LIN {X 0,Y 67.395,Z 528.799,A -85,B 0,C 180,E1 -28557.992,E2 -28557.992} C_VEL
LIN {X 0,Y 71.821,Z 521.872,A -85,B 0,C 180,E1 -28565.959,E2 -28565.959} C_VEL
LIN {X 0,Y 75.45,Z 516.289,A -85,B 0,C 180,E1 -28570.701,E2 -28570.701} C_VEL
LIN {X 0,Y 79.441,Z 509.825,A -85,B 0,C 180,E1 -28575.058,E2 -28575.058} C_VEL
LIN {X 0,Y 85.076,Z 500.094,A -85,B 0,C 180,E1 -28579.836,E2 -28579.836} C_VEL
LIN {X 0,Y 90.563,Z 489.267,A -85,B 0,C 180,E1 -28583.63,E2 -28583.63} C_VEL
LIN {X 0,Y 95.195,Z 478.806,A -85,B 0,C 180,E1 -28586.162,E2 -28586.162} C_VEL
LIN {X 0,Y 99.231,Z 467.304,A -85,B 0,C 180,E1 -28588.207,E2 -28588.207} C_VEL
LIN {X 0,Y 102.796,Z 453.682,A -85,B 0,C 180,E1 -28589.877,E2 -28589.877} C_VEL
LIN {X 0,Y 105.087,Z 440.795,A -85,B 0,C 180,E1 -28590.836,E2 -28590.836} C_VEL
LIN {X 0,Y 108.243,Z 407.199,A -85,B 0,C 180,E1 -28592.444,E2 -28592.444} C_VEL
LIN {X 0,Y 106.476,Z 400.809,A -85,B 0,C 180,E1 -28594.667,E2 -28594.667} C_VEL
LIN {X 0,Y 103.203,Z 393.621,A -85,B 0,C 180,E1 -28598.746,E2 -28598.746} C_VEL
LIN {X 0,Y 100.195,Z 388.023,A -85,B 0,C 180,E1 -28603.115,E2 -28603.115} C_VEL
LIN {X 0,Y 98.336,Z 384.757,A -85,B 0,C 180,E1 -28606.346,E2 -28606.346} C_VEL
LIN {X 0,Y 96.433,Z 381.395,A -85,B 0,C 180,E1 -28610.429,E2 -28610.429} C_VEL
LIN {X 0,Y 94.56,Z 377.804,A -85,B 0,C 180,E1 -28616.137,E2 -28616.137} C_VEL
LIN {X 0,Y 94.415,Z 377.342,A -85,B 0,C 180,E1 -28616.799,E2 -28616.799} C_VEL
LIN {X 0,Y 93.361,Z 376.43,A -85,B 0,C 180,E1 -28622.156,E2 -28622.156} C_VEL
LIN {X 0,Y 93.22,Z 376.695,A -85,B 0,C 180,E1 -28631.436,E2 -28631.436} C_VEL
LIN {X 0,Y 94.275,Z 377.725,A -85,B 0,C 180,E1 -28637.348,E2 -28637.348} C_VEL
LIN {X 0,Y 94.428,Z 378.267,A -85,B 0,C 180,E1 -28638.09,E2 -28638.09} C_VEL
LIN {X 0,Y 95.513,Z 382.03,A -85,B 0,C 180,E1 -28642.263,E2 -28642.263} C_VEL
LIN {X 0,Y 96.776,Z 386.789,A -85,B 0,C 180,E1 -28646,E2 -28646} C_VEL
LIN {X 0,Y 99.897,Z 397.718,A -85,B 0,C 180,E1 -28652.646,E2 -28652.646} C_VEL
LIN {X 0,Y 103.176,Z 405.13,A -85,B 0,C 180,E1 -28657.343,E2 -28657.343} C_VEL
LIN {X 0,Y 104.285,Z 408.071,A -85,B 0,C 180,E1 -28658.794,E2 -28658.794} C_VEL
LIN {X 0,Y 100.967,Z 439.433,A -85,B 0,C 180,E1 -28660.188,E2 -28660.188} C_VEL
LIN {X 0,Y 98.399,Z 452.745,A -85,B 0,C 180,E1 -28661.288,E2 -28661.288} C_VEL
LIN {X 0,Y 94.745,Z 465.531,A -85,B 0,C 180,E1 -28662.898,E2 -28662.898} C_VEL
LIN {X 0,Y 90.061,Z 478.114,A -85,B 0,C 180,E1 -28665.381,E2 -28665.381} C_VEL
LIN {X 0,Y 84.771,Z 489.367,A -85,B 0,C 180,E1 -28668.447,E2 -28668.447} C_VEL
LIN {X 0,Y 79.094,Z 499.489,A -85,B 0,C 180,E1 -28672.341,E2 -28672.341} C_VEL
LIN {X 0,Y 72.715,Z 509.449,A -85,B 0,C 180,E1 -28677.882,E2 -28677.882} C_VEL
LIN {X 0,Y 67.524,Z 516.86,A -85,B 0,C 180,E1 -28683.741,E2 -28683.741} C_VEL
LIN {X 0,Y 62.326,Z 524.149,A -85,B 0,C 180,E1 -28691.929,E2 -28691.929} C_VEL
LIN {X 0,Y 59.034,Z 529.063,A -85,B 0,C 180,E1 -28699.707,E2 -28699.707} C_VEL
LIN {X 0,Y 56.229,Z 534.211,A -85,B 0,C 180,E1 -28710.881,E2 -28710.881} C_VEL
LIN {X 0,Y 55.041,Z 537.544,A -85,B 0,C 180,E1 -28721.035,E2 -28721.035} C_VEL
LIN {X 0,Y 55.546,Z 540.194,A -85,B 0,C 180,E1 -28732.3,E2 -28732.3} C_VEL
LIN {X 0,Y 57.124,Z 541.55,A -85,B 0,C 180,E1 -28740.55,E2 -28740.55} C_VEL
LIN {X 0,Y 61.757,Z 542.59,A -85,B 0,C 180,E1 -28753.055,E2 -28753.055} C_VEL
LIN {X 0,Y 66.593,Z 542.434,A -85,B 0,C 180,E1 -28760.714,E2 -28760.714} C_VEL
LIN {X 0,Y 73.958,Z 541.167,A -85,B 0,C 180,E1 -28768.776,E2 -28768.776} C_VEL
LIN {X 0,Y 81.078,Z 539.175,A -85,B 0,C 180,E1 -28774.317,E2 -28774.317} C_VEL
LIN {X 0,Y 89.982,Z 535.765,A -85,B 0,C 180,E1 -28779.583,E2 -28779.583} C_VEL
LIN {X 0,Y 99.493,Z 531.064,A -85,B 0,C 180,E1 -28783.882,E2 -28783.882} C_VEL
LIN {X 0,Y 109.778,Z 524.705,A -85,B 0,C 180,E1 -28787.486,E2 -28787.486} C_VEL
LIN {X 0,Y 119.877,Z 516.921,A -85,B 0,C 180,E1 -28790.279,E2 -28790.279} C_VEL
LIN {X 0,Y 129.367,Z 507.98,A -85,B 0,C 180,E1 -28792.477,E2 -28792.477} C_VEL
LIN {X 0,Y 137.79,Z 498.207,A -85,B 0,C 180,E1 -28794.146,E2 -28794.146} C_VEL
LIN {X 0,Y 145.397,Z 487.356,A -85,B 0,C 180,E1 -28795.483,E2 -28795.483} C_VEL
LIN {X 0,Y 151.388,Z 476.779,A -85,B 0,C 180,E1 -28796.431,E2 -28796.431} C_VEL
LIN {X 0,Y 156.602,Z 465.018,A -85,B 0,C 180,E1 -28797.232,E2 -28797.232} C_VEL
LIN {X 0,Y 159.81,Z 455.577,A -85,B 0,C 180,E1 -28797.795,E2 -28797.795} C_VEL
LIN {X 0,Y 159.495,Z 453.125,A -85,B 0,C 180,E1 -28800.632,E2 -28800.632} C_VEL
LIN {X 0,Y 159.412,Z 451.352,A -85,B 0,C 180,E1 -28803.16,E2 -28803.16} C_VEL
LIN {X 0,Y 159.249,Z 451.359,A -85,B 0,C 180,E1 -28808.886,E2 -28808.886} C_VEL
LIN {X 0,Y 159.381,Z 451.899,A -85,B 0,C 180,E1 -28810.641,E2 -28810.641} C_VEL
LIN {X 0,Y 159.89,Z 455.058,A -85,B 0,C 180,E1 -28815.137,E2 -28815.137} C_VEL
LIN {X 0,Y 159.936,Z 455.914,A -85,B 0,C 180,E1 -28815.799,E2 -28815.799} C_VEL
LIN {X 0,Y 158.991,Z 459.189,A -85,B 0,C 180,E1 -28816.092,E2 -28816.092} C_VEL
LIN {X 0,Y 154.069,Z 472.123,A -85,B 0,C 180,E1 -28816.687,E2 -28816.687} C_VEL
LIN {X 0,Y 148.232,Z 483.649,A -85,B 0,C 180,E1 -28817.423,E2 -28817.423} C_VEL
LIN {X 0,Y 140.817,Z 495.255,A -85,B 0,C 180,E1 -28818.52,E2 -28818.52} C_VEL
LIN {X 0,Y 132.693,Z 505.572,A -85,B 0,C 180,E1 -28819.938,E2 -28819.938} C_VEL
LIN {X 0,Y 124.643,Z 513.958,A -85,B 0,C 180,E1 -28821.519,E2 -28821.519} C_VEL
LIN {X 0,Y 115.178,Z 522.163,A -85,B 0,C 180,E1 -28823.763,E2 -28823.763} C_VEL
LIN {X 0,Y 105.915,Z 528.799,A -85,B 0,C 180,E1 -28826.398,E2 -28826.398} C_VEL
LIN {X 0,Y 96.935,Z 534.118,A -85,B 0,C 180,E1 -28829.546,E2 -28829.546} C_VEL
LIN {X 0,Y 88.467,Z 538.285,A -85,B 0,C 180,E1 -28833.481,E2 -28833.481} C_VEL
LIN {X 0,Y 80.522,Z 541.427,A -85,B 0,C 180,E1 -28838.239,E2 -28838.239} C_VEL
LIN {X 0,Y 75.531,Z 543.01,A -85,B 0,C 180,E1 -28841.902,E2 -28841.902} C_VEL
LIN {X 0,Y 70.922,Z 544.187,A -85,B 0,C 180,E1 -28846.087,E2 -28846.087} C_VEL
LIN {X 0,Y 63.079,Z 545.327,A -85,B 0,C 180,E1 -28856.153,E2 -28856.153} C_VEL
LIN {X 0,Y 57.904,Z 544.98,A -85,B 0,C 180,E1 -28868.653,E2 -28868.653} C_VEL
LIN {X 0,Y 56.397,Z 544.201,A -85,B 0,C 180,E1 -28875.575,E2 -28875.575} C_VEL
LIN {X 0,Y 55.666,Z 543.021,A -85,B 0,C 180,E1 -28882.753,E2 -28882.753} C_VEL
LIN {X 0,Y 55.585,Z 541.436,A -85,B 0,C 180,E1 -28890.007,E2 -28890.007} C_VEL
LIN {X 0,Y 55.884,Z 538.153,A -85,B 0,C 180,E1 -28900.88,E2 -28900.88} C_VEL
LIN {X 0,Y 57.696,Z 533.757,A -85,B 0,C 180,E1 -28911.441,E2 -28911.441} C_VEL
LIN {X 0,Y 61.189,Z 528.137,A -85,B 0,C 180,E1 -28921.128,E2 -28921.128} C_VEL
LIN {X 0,Y 66.145,Z 521.09,A -85,B 0,C 180,E1 -28929.613,E2 -28929.613} C_VEL
LIN {X 0,Y 70.855,Z 514.227,A -85,B 0,C 180,E1 -28935.509,E2 -28935.509} C_VEL
LIN {X 0,Y 76.943,Z 505.107,A -85,B 0,C 180,E1 -28940.938,E2 -28940.938} C_VEL
LIN {X 0,Y 82.565,Z 495.477,A -85,B 0,C 180,E1 -28945.021,E2 -28945.021} C_VEL
LIN {X 0,Y 86.552,Z 487.852,A -85,B 0,C 180,E1 -28947.407,E2 -28947.407} C_VEL
LIN {X 0,Y 91.371,Z 476.986,A -85,B 0,C 180,E1 -28949.926,E2 -28949.926} C_VEL
LIN {X 0,Y 95.634,Z 465.013,A -85,B 0,C 180,E1 -28951.875,E2 -28951.875} C_VEL
LIN {X 0,Y 99.053,Z 452.141,A -85,B 0,C 180,E1 -28953.302,E2 -28953.302} C_VEL
LIN {X 0,Y 101.283,Z 439.357,A -85,B 0,C 180,E1 -28954.149,E2 -28954.149} C_VEL
LIN {X 0,Y 104.193,Z 409.232,A -85,B 0,C 180,E1 -28955.597,E2 -28955.597} C_VEL
LIN {X 0,Y 103.128,Z 405.212,A -85,B 0,C 180,E1 -28957.153,E2 -28957.153} C_VEL
LIN {X 0,Y 100.484,Z 398.932,A -85,B 0,C 180,E1 -28960.927,E2 -28960.927} C_VEL
LIN {X 0,Y 97.838,Z 393.623,A -85,B 0,C 180,E1 -28965.311,E2 -28965.311} C_VEL
LIN {X 0,Y 96.248,Z 390.603,A -85,B 0,C 180,E1 -28968.515,E2 -28968.515} C_VEL
LIN {X 0,Y 94.886,Z 387.929,A -85,B 0,C 180,E1 -28971.9,E2 -28971.9} C_VEL
LIN {X 0,Y 93.251,Z 384.228,A -85,B 0,C 180,E1 -28977.839,E2 -28977.839} C_VEL
LIN {X 0,Y 92.476,Z 383.477,A -85,B 0,C 180,E1 -28982.177,E2 -28982.177} C_VEL
LIN {X 0,Y 92.233,Z 383.622,A -85,B 0,C 180,E1 -28990.16,E2 -28990.16} C_VEL
LIN {X 0,Y 93.141,Z 384.688,A -85,B 0,C 180,E1 -28996.418,E2 -28996.418} C_VEL
LIN {X 0,Y 94.834,Z 388.195,A -85,B 0,C 180,E1 -29002.524,E2 -29002.524} C_VEL
LIN {X 0,Y 97.347,Z 392.63,A -85,B 0,C 180,E1 -29008.217,E2 -29008.217} C_VEL
LIN {X 0,Y 99.897,Z 397.718,A -85,B 0,C 180,E1 -29012.646,E2 -29012.646} C_VEL
LIN {X 0,Y 100.591,Z 400.78,A -85,B 0,C 180,E1 -29013.964,E2 -29013.964} C_VEL
LIN {X 0,Y 100.925,Z 404.327,A -85,B 0,C 180,E1 -29014.89,E2 -29014.89} C_VEL
LIN {X 0,Y 100.874,Z 410.12,A -85,B 0,C 180,E1 -29015.712,E2 -29015.712} C_VEL
LIN {X 0,Y 99.782,Z 420.474,A -85,B 0,C 180,E1 -29016.109,E2 -29016.109} C_VEL
LIN {X 0,Y 98.669,Z 428.86,A -85,B 0,C 180,E1 -29016.193,E2 -29016.193} C_VEL
LIN {X 0,Y 96.727,Z 443.461,A -85,B 0,C 180,E1 -29016.937,E2 -29016.937} C_VEL
LIN {X 0,Y 94.117,Z 455.135,A -85,B 0,C 180,E1 -29017.954,E2 -29017.954} C_VEL
LIN {X 0,Y 90.063,Z 467.848,A -85,B 0,C 180,E1 -29019.587,E2 -29019.587} C_VEL
LIN {X 0,Y 85.173,Z 479.992,A -85,B 0,C 180,E1 -29022.038,E2 -29022.038} C_VEL
LIN {X 0,Y 79.607,Z 490.864,A -85,B 0,C 180,E1 -29025.062,E2 -29025.062} C_VEL
LIN {X 0,Y 72.927,Z 501.718,A -85,B 0,C 180,E1 -29029.415,E2 -29029.415} C_VEL
LIN {X 0,Y 66.781,Z 510.521,A -85,B 0,C 180,E1 -29034.626,E2 -29034.626} C_VEL
LIN {X 0,Y 61.203,Z 517.786,A -85,B 0,C 180,E1 -29040.782,E2 -29040.782} C_VEL
LIN {X 0,Y 55.586,Z 524.912,A -85,B 0,C 180,E1 -29049.647,E2 -29049.647} C_VEL
LIN {X 0,Y 51.988,Z 529.751,A -85,B 0,C 180,E1 -29058.294,E2 -29058.294} C_VEL
LIN {X 0,Y 49.157,Z 534.438,A -85,B 0,C 180,E1 -29069.993,E2 -29069.993} C_VEL
LIN {X 0,Y 47.905,Z 538.037,A -85,B 0,C 180,E1 -29082.705,E2 -29082.705} C_VEL
LIN {X 0,Y 48.813,Z 540.599,A -85,B 0,C 180,E1 -29095.582,E2 -29095.582} C_VEL
LIN {X 0,Y 50.603,Z 541.752,A -85,B 0,C 180,E1 -29103.739,E2 -29103.739} C_VEL
LIN {X 0,Y 53.166,Z 542.487,A -85,B 0,C 180,E1 -29111.363,E2 -29111.363} C_VEL
LIN {X 0,Y 56.571,Z 542.818,A -85,B 0,C 180,E1 -29118.183,E2 -29118.183} C_VEL
LIN {X 0,Y 61.298,Z 542.664,A -85,B 0,C 180,E1 -29125.024,E2 -29125.024} C_VEL
LIN {X 0,Y 70.383,Z 541.225,A -85,B 0,C 180,E1 -29133.973,E2 -29133.973} C_VEL
LIN {X 0,Y 77.162,Z 539.457,A -85,B 0,C 180,E1 -29138.635,E2 -29138.635} C_VEL
LIN {X 0,Y 87.665,Z 535.643,A -85,B 0,C 180,E1 -29144.143,E2 -29144.143} C_VEL
LIN {X 0,Y 97.093,Z 531.155,A -85,B 0,C 180,E1 -29147.854,E2 -29147.854} C_VEL
LIN {X 0,Y 106.766,Z 525.433,A -85,B 0,C 180,E1 -29150.867,E2 -29150.867} C_VEL
LIN {X 0,Y 115.369,Z 519.264,A -85,B 0,C 180,E1 -29153.003,E2 -29153.003} C_VEL
LIN {X 0,Y 123.497,Z 512.305,A -85,B 0,C 180,E1 -29154.768,E2 -29154.768} C_VEL
LIN {X 0,Y 132.039,Z 503.574,A -85,B 0,C 180,E1 -29156.327,E2 -29156.327} C_VEL
LIN {X 0,Y 140.661,Z 492.676,A -85,B 0,C 180,E1 -29157.746,E2 -29157.746} C_VEL
LIN {X 0,Y 147.617,Z 481.805,A -85,B 0,C 180,E1 -29158.727,E2 -29158.727} C_VEL
LIN {X 0,Y 153.416,Z 470.274,A -85,B 0,C 180,E1 -29159.529,E2 -29159.529} C_VEL
LIN {X 0,Y 157.006,Z 461.289,A -85,B 0,C 180,E1 -29160.001,E2 -29160.001} C_VEL
LIN {X 0,Y 157.23,Z 459.607,A -85,B 0,C 180,E1 -29161.281,E2 -29161.281} C_VEL
LIN {X 0,Y 157.225,Z 458.761,A -85,B 0,C 180,E1 -29162.563,E2 -29162.563} C_VEL
LIN {X 0,Y 157.14,Z 457.986,A -85,B 0,C 180,E1 -29165.133,E2 -29165.133} C_VEL
LIN {X 0,Y 157.116,Z 458.026,A -85,B 0,C 180,E1 -29167.713,E2 -29167.713} C_VEL
LIN {X 0,Y 157.236,Z 458.773,A -85,B 0,C 180,E1 -29170.49,E2 -29170.49} C_VEL
LIN {X 0,Y 157.387,Z 460.515,A -85,B 0,C 180,E1 -29173.263,E2 -29173.263} C_VEL
LIN {X 0,Y 156.973,Z 462.087,A -85,B 0,C 180,E1 -29173.648,E2 -29173.648} C_VEL
LIN {X 0,Y 152.198,Z 473.668,A -85,B 0,C 180,E1 -29174.15,E2 -29174.15} C_VEL
LIN {X 0,Y 146.274,Z 484.818,A -85,B 0,C 180,E1 -29174.785,E2 -29174.785} C_VEL
LIN {X 0,Y 138.74,Z 496.182,A -85,B 0,C 180,E1 -29175.76,E2 -29175.76} C_VEL
LIN {X 0,Y 130.456,Z 506.233,A -85,B 0,C 180,E1 -29177.023,E2 -29177.023} C_VEL
LIN {X 0,Y 123.852,Z 512.978,A -85,B 0,C 180,E1 -29178.117,E2 -29178.117} C_VEL
LIN {X 0,Y 114.113,Z 521.332,A -85,B 0,C 180,E1 -29180.09,E2 -29180.09} C_VEL
LIN {X 0,Y 104.54,Z 528.08,A -85,B 0,C 180,E1 -29182.435,E2 -29182.435} C_VEL
LIN {X 0,Y 93.646,Z 534.308,A -85,B 0,C 180,E1 -29185.775,E2 -29185.775} C_VEL
LIN {X 0,Y 84.75,Z 538.385,A -85,B 0,C 180,E1 -29189.466,E2 -29189.466} C_VEL
LIN {X 0,Y 76.315,Z 541.443,A -85,B 0,C 180,E1 -29194.031,E2 -29194.031} C_VEL
LIN {X 0,Y 70.984,Z 542.982,A -85,B 0,C 180,E1 -29197.63,E2 -29197.63} C_VEL
LIN {X 0,Y 61.402,Z 544.803,A -85,B 0,C 180,E1 -29206.635,E2 -29206.635} C_VEL
LIN {X 0,Y 53.937,Z 545.122,A -85,B 0,C 180,E1 -29218.595,E2 -29218.595} C_VEL
LIN {X 0,Y 51.344,Z 544.704,A -85,B 0,C 180,E1 -29225.763,E2 -29225.763} C_VEL
LIN {X 0,Y 48.62,Z 542.656,A -85,B 0,C 180,E1 -29241.697,E2 -29241.697} C_VEL
LIN {X 0,Y 48.485,Z 541.033,A -85,B 0,C 180,E1 -29250.008,E2 -29250.008} C_VEL
LIN {X 0,Y 48.928,Z 537.671,A -85,B 0,C 180,E1 -29262.45,E2 -29262.45} C_VEL
LIN {X 0,Y 51.107,Z 533.186,A -85,B 0,C 180,E1 -29274.373,E2 -29274.373} C_VEL
LIN {X 0,Y 55.187,Z 527.472,A -85,B 0,C 180,E1 -29284.972,E2 -29284.972} C_VEL
LIN {X 0,Y 60.802,Z 520.27,A -85,B 0,C 180,E1 -29293.918,E2 -29293.918} C_VEL
LIN {X 0,Y 65.15,Z 514.498,A -85,B 0,C 180,E1 -29299.044,E2 -29299.044} C_VEL
LIN {X 0,Y 71.37,Z 505.978,A -85,B 0,C 180,E1 -29304.34,E2 -29304.34} C_VEL
LIN {X 0,Y 77.315,Z 496.576,A -85,B 0,C 180,E1 -29308.46,E2 -29308.46} C_VEL
LIN {X 0,Y 81.459,Z 489.102,A -85,B 0,C 180,E1 -29310.882,E2 -29310.882} C_VEL
LIN {X 0,Y 86.564,Z 478.697,A -85,B 0,C 180,E1 -29313.271,E2 -29313.271} C_VEL
LIN {X 0,Y 91.003,Z 467.314,A -85,B 0,C 180,E1 -29315.162,E2 -29315.162} C_VEL
LIN {X 0,Y 94.921,Z 453.666,A -85,B 0,C 180,E1 -29316.731,E2 -29316.731} C_VEL
LIN {X 0,Y 97.433,Z 440.946,A -85,B 0,C 180,E1 -29317.588,E2 -29317.588} C_VEL
LIN {X 0,Y 100.54,Z 411.619,A -85,B 0,C 180,E1 -29318.878,E2 -29318.878} C_VEL
LIN {X 0,Y 99.737,Z 408.886,A -85,B 0,C 180,E1 -29320.193,E2 -29320.193} C_VEL
LIN {X 0,Y 97.316,Z 402.878,A -85,B 0,C 180,E1 -29324.272,E2 -29324.272} C_VEL
LIN {X 0,Y 94.937,Z 397.665,A -85,B 0,C 180,E1 -29329.216,E2 -29329.216} C_VEL
LIN {X 0,Y 93.317,Z 394.285,A -85,B 0,C 180,E1 -29333.702,E2 -29333.702} C_VEL
LIN {X 0,Y 92.034,Z 391.003,A -85,B 0,C 180,E1 -29339.349,E2 -29339.349} C_VEL
LIN {X 0,Y 91.37,Z 390.438,A -85,B 0,C 180,E1 -29344.41,E2 -29344.41} C_VEL
LIN {X 0,Y 91.567,Z 390.965,A -85,B 0,C 180,E1 -29352.468,E2 -29352.468} C_VEL
LIN {X 0,Y 92.013,Z 391.551,A -85,B 0,C 180,E1 -29355.321,E2 -29355.321} C_VEL
LIN {X 0,Y 93.859,Z 395.689,A -85,B 0,C 180,E1 -29362.509,E2 -29362.509} C_VEL
LIN {X 0,Y 95.883,Z 399.776,A -85,B 0,C 180,E1 -29367.398,E2 -29367.398} C_VEL
LIN {X 0,Y 98.266,Z 405.159,A -85,B 0,C 180,E1 -29371.887,E2 -29371.887} C_VEL
LIN {X 0,Y 100.492,Z 410.819,A -85,B 0,C 180,E1 -29375.411,E2 -29375.411} C_VEL
LIN {X 0,Y 98.669,Z 428.86,A -85,B 0,C 180,E1 -29376.193,E2 -29376.193} C_VEL
LIN {X 0,Y 97.631,Z 434.674,A -85,B 0,C 180,E1 -29376.007,E2 -29376.007} C_VEL
LIN {X 0,Y 94.822,Z 444.034,A -85,B 0,C 180,E1 -29374.985,E2 -29374.985} C_VEL
LIN {X 0,Y 91.478,Z 453.259,A -85,B 0,C 180,E1 -29374.199,E2 -29374.199} C_VEL
LIN {X 0,Y 89.626,Z 458.855,A -85,B 0,C 180,E1 -29374.43,E2 -29374.43} C_VEL
LIN {X 0,Y 85.717,Z 470.062,A -85,B 0,C 180,E1 -29375.931,E2 -29375.931} C_VEL
LIN {X 0,Y 80.611,Z 481.692,A -85,B 0,C 180,E1 -29378.304,E2 -29378.304} C_VEL
LIN {X 0,Y 74.472,Z 492.694,A -85,B 0,C 180,E1 -29381.344,E2 -29381.344} C_VEL
LIN {X 0,Y 67.69,Z 502.914,A -85,B 0,C 180,E1 -29385.5,E2 -29385.5} C_VEL
LIN {X 0,Y 61.092,Z 511.537,A -85,B 0,C 180,E1 -29390.742,E2 -29390.742} C_VEL
LIN {X 0,Y 53.957,Z 519.909,A -85,B 0,C 180,E1 -29398.593,E2 -29398.593} C_VEL
LIN {X 0,Y 48.108,Z 526.646,A -85,B 0,C 180,E1 -29408.571,E2 -29408.571} C_VEL
LIN {X 0,Y 43.796,Z 532.033,A -85,B 0,C 180,E1 -29420.757,E2 -29420.757} C_VEL
LIN {X 0,Y 41.269,Z 536.259,A -85,B 0,C 180,E1 -29434.876,E2 -29434.876} C_VEL
LIN {X 0,Y 40.999,Z 539.419,A -85,B 0,C 180,E1 -29450.04,E2 -29450.04} C_VEL
LIN {X 0,Y 44.025,Z 541.872,A -85,B 0,C 180,E1 -29467.047,E2 -29467.047} C_VEL
LIN {X 0,Y 47.841,Z 542.758,A -85,B 0,C 180,E1 -29477.255,E2 -29477.255} C_VEL
LIN {X 0,Y 51.913,Z 543.046,A -85,B 0,C 180,E1 -29484.307,E2 -29484.307} C_VEL
LIN {X 0,Y 56.614,Z 542.876,A -85,B 0,C 180,E1 -29490.326,E2 -29490.326} C_VEL
LIN {X 0,Y 61.835,Z 542.284,A -85,B 0,C 180,E1 -29495.389,E2 -29495.389} C_VEL
LIN {X 0,Y 67.457,Z 541.283,A -85,B 0,C 180,E1 -29499.645,E2 -29499.645} C_VEL
LIN {X 0,Y 73.708,Z 539.745,A -85,B 0,C 180,E1 -29503.38,E2 -29503.38} C_VEL
LIN {X 0,Y 82.728,Z 536.789,A -85,B 0,C 180,E1 -29507.655,E2 -29507.655} C_VEL
LIN {X 0,Y 92.783,Z 532.444,A -85,B 0,C 180,E1 -29511.288,E2 -29511.288} C_VEL
LIN {X 0,Y 104.149,Z 526.141,A -85,B 0,C 180,E1 -29514.424,E2 -29514.424} C_VEL
LIN {X 0,Y 113.607,Z 519.627,A -85,B 0,C 180,E1 -29516.454,E2 -29516.454} C_VEL
LIN {X 0,Y 123.044,Z 511.704,A -85,B 0,C 180,E1 -29518.186,E2 -29518.186} C_VEL
LIN {X 0,Y 132.649,Z 501.748,A -85,B 0,C 180,E1 -29519.643,E2 -29519.643} C_VEL
LIN {X 0,Y 140.564,Z 491.649,A -85,B 0,C 180,E1 -29520.733,E2 -29520.733} C_VEL
LIN {X 0,Y 147.636,Z 480.403,A -85,B 0,C 180,E1 -29521.575,E2 -29521.575} C_VEL
LIN {X 0,Y 153.325,Z 468.871,A -85,B 0,C 180,E1 -29522.246,E2 -29522.246} C_VEL
LIN {X 0,Y 154.284,Z 466.654,A -85,B 0,C 180,E1 -29522.358,E2 -29522.358} C_VEL
LIN {X 0,Y 154.689,Z 465.541,A -85,B 0,C 180,E1 -29522.605,E2 -29522.605} C_VEL
LIN {X 0,Y 154.7,Z 464.668,A -85,B 0,C 180,E1 -29525.214,E2 -29525.214} C_VEL
LIN {X 0,Y 154.688,Z 464.737,A -85,B 0,C 180,E1 -29527.834,E2 -29527.834} C_VEL
LIN {X 0,Y 154.72,Z 465.589,A -85,B 0,C 180,E1 -29530.469,E2 -29530.469} C_VEL
LIN {X 0,Y 154.145,Z 467.442,A -85,B 0,C 180,E1 -29531.248,E2 -29531.248} C_VEL
LIN {X 0,Y 148.056,Z 480.102,A -85,B 0,C 180,E1 -29531.765,E2 -29531.765} C_VEL
LIN {X 0,Y 141.246,Z 491.215,A -85,B 0,C 180,E1 -29532.465,E2 -29532.465} C_VEL
LIN {X 0,Y 133.619,Z 501.249,A -85,B 0,C 180,E1 -29533.346,E2 -29533.346} C_VEL
LIN {X 0,Y 125.177,Z 510.329,A -85,B 0,C 180,E1 -29534.434,E2 -29534.434} C_VEL
LIN {X 0,Y 115.2,Z 519.181,A -85,B 0,C 180,E1 -29536.096,E2 -29536.096} C_VEL
LIN {X 0,Y 105.299,Z 526.338,A -85,B 0,C 180,E1 -29538.006,E2 -29538.006} C_VEL
LIN {X 0,Y 93.968,Z 532.885,A -85,B 0,C 180,E1 -29540.801,E2 -29540.801} C_VEL
LIN {X 0,Y 84.543,Z 537.242,A -85,B 0,C 180,E1 -29543.888,E2 -29543.888} C_VEL
LIN {X 0,Y 72.569,Z 541.46,A -85,B 0,C 180,E1 -29549.364,E2 -29549.364} C_VEL
LIN {X 0,Y 66.884,Z 542.928,A -85,B 0,C 180,E1 -29552.805,E2 -29552.805} C_VEL
LIN {X 0,Y 56.441,Z 544.662,A -85,B 0,C 180,E1 -29561.669,E2 -29561.669} C_VEL
LIN {X 0,Y 47.989,Z 544.893,A -85,B 0,C 180,E1 -29574.15,E2 -29574.15} C_VEL
LIN {X 0,Y 44.958,Z 544.408,A -85,B 0,C 180,E1 -29582.042,E2 -29582.042} C_VEL
LIN {X 0,Y 41.61,Z 542.286,A -85,B 0,C 180,E1 -29600.285,E2 -29600.285} C_VEL
LIN {X 0,Y 41.403,Z 540.622,A -85,B 0,C 180,E1 -29610.009,E2 -29610.009} C_VEL
LIN {X 0,Y 42.005,Z 537.179,A -85,B 0,C 180,E1 -29624.544,E2 -29624.544} C_VEL
LIN {X 0,Y 44.702,Z 532.603,A -85,B 0,C 180,E1 -29638.151,E2 -29638.151} C_VEL
LIN {X 0,Y 50.525,Z 525.641,A -85,B 0,C 180,E1 -29651.365,E2 -29651.365} C_VEL
LIN {X 0,Y 57.093,Z 518.063,A -85,B 0,C 180,E1 -29660.306,E2 -29660.306} C_VEL
LIN {X 0,Y 63.108,Z 510.574,A -85,B 0,C 180,E1 -29666.162,E2 -29666.162} C_VEL
LIN {X 0,Y 69.513,Z 501.885,A -85,B 0,C 180,E1 -29670.703,E2 -29670.703} C_VEL
LIN {X 0,Y 75.223,Z 492.852,A -85,B 0,C 180,E1 -29674.069,E2 -29674.069} C_VEL
LIN {X 0,Y 81.314,Z 481.793,A -85,B 0,C 180,E1 -29676.693,E2 -29676.693} C_VEL
LIN {X 0,Y 85.899,Z 471.315,A -85,B 0,C 180,E1 -29678.55,E2 -29678.55} C_VEL
LIN {X 0,Y 90.164,Z 458.818,A -85,B 0,C 180,E1 -29680.063,E2 -29680.063} C_VEL
LIN {X 0,Y 93.262,Z 445.957,A -85,B 0,C 180,E1 -29681.099,E2 -29681.099} C_VEL
LIN {X 0,Y 95.277,Z 431.774,A -85,B 0,C 180,E1 -29681.731,E2 -29681.731} C_VEL
LIN {X 0,Y 97.115,Z 414.225,A -85,B 0,C 180,E1 -29682.467,E2 -29682.467} C_VEL
LIN {X 0,Y 95.134,Z 408.658,A -85,B 0,C 180,E1 -29686.372,E2 -29686.372} C_VEL
LIN {X 0,Y 93.167,Z 403.796,A -85,B 0,C 180,E1 -29691.168,E2 -29691.168} C_VEL
LIN {X 0,Y 91.923,Z 400.743,A -85,B 0,C 180,E1 -29695.28,E2 -29695.28} C_VEL
LIN {X 0,Y 90.935,Z 397.842,A -85,B 0,C 180,E1 -29700.552,E2 -29700.552} C_VEL
LIN {X 0,Y 90.489,Z 397.473,A -85,B 0,C 180,E1 -29704.453,E2 -29704.453} C_VEL
LIN {X 0,Y 90.812,Z 398.169,A -85,B 0,C 180,E1 -29713.424,E2 -29713.424} C_VEL
LIN {X 0,Y 92.391,Z 402.215,A -85,B 0,C 180,E1 -29720.996,E2 -29720.996} C_VEL
LIN {X 0,Y 93.998,Z 405.88,A -85,B 0,C 180,E1 -29725.509,E2 -29725.509} C_VEL
LIN {X 0,Y 96.103,Z 411.265,A -85,B 0,C 180,E1 -29730.085,E2 -29730.085} C_VEL
LIN {X 0,Y 97.02,Z 413.872,A -85,B 0,C 180,E1 -29731.819,E2 -29731.819} C_VEL
LIN {X 0,Y 95.48,Z 428.661,A -85,B 0,C 180,E1 -29732.452,E2 -29732.452} C_VEL
LIN {X 0,Y 93.449,Z 443.424,A -85,B 0,C 180,E1 -29733.134,E2 -29733.134} C_VEL
LIN {X 0,Y 90.583,Z 455.707,A -85,B 0,C 180,E1 -29734.133,E2 -29734.133} C_VEL
LIN {X 0,Y 89.626,Z 458.855,A -85,B 0,C 180,E1 -29734.43,E2 -29734.43} C_VEL
LIN {X 0,Y 87.558,Z 464.379,A -85,B 0,C 180,E1 -29734.692,E2 -29734.692} C_VEL
LIN {X 0,Y 82.929,Z 473.129,A -85,B 0,C 180,E1 -29734.33,E2 -29734.33} C_VEL
LIN {X 0,Y 77.672,Z 481.535,A -85,B 0,C 180,E1 -29734.149,E2 -29734.149} C_VEL
LIN {X 0,Y 74.618,Z 486.524,A -85,B 0,C 180,E1 -29734.818,E2 -29734.818} C_VEL
LIN {X 0,Y 67.991,Z 497.009,A -85,B 0,C 180,E1 -29737.977,E2 -29737.977} C_VEL
LIN {X 0,Y 61.38,Z 505.859,A -85,B 0,C 180,E1 -29741.897,E2 -29741.897} C_VEL
LIN {X 0,Y 54.377,Z 514,A -85,B 0,C 180,E1 -29747.262,E2 -29747.262} C_VEL
LIN {X 0,Y 46.799,Z 521.976,A -85,B 0,C 180,E1 -29755.717,E2 -29755.717} C_VEL
LIN {X 0,Y 41.519,Z 527.363,A -85,B 0,C 180,E1 -29764.955,E2 -29764.955} C_VEL
LIN {X 0,Y 36.709,Z 532.649,A -85,B 0,C 180,E1 -29778.952,E2 -29778.952} C_VEL
LIN {X 0,Y 34.003,Z 536.784,A -85,B 0,C 180,E1 -29795.921,E2 -29795.921} C_VEL
LIN {X 0,Y 34.196,Z 539.857,A -85,B 0,C 180,E1 -29814.259,E2 -29814.259} C_VEL
LIN {X 0,Y 37.804,Z 542.028,A -85,B 0,C 180,E1 -29831.962,E2 -29831.962} C_VEL
LIN {X 0,Y 43.161,Z 543.029,A -85,B 0,C 180,E1 -29844.49,E2 -29844.49} C_VEL
LIN {X 0,Y 52.079,Z 543.123,A -85,B 0,C 180,E1 -29856.12,E2 -29856.12} C_VEL
LIN {X 0,Y 59.12,Z 542.385,A -85,B 0,C 180,E1 -29861.97,E2 -29861.97} C_VEL
LIN {X 0,Y 65.245,Z 541.338,A -85,B 0,C 180,E1 -29865.778,E2 -29865.778} C_VEL
LIN {X 0,Y 71.609,Z 539.806,A -85,B 0,C 180,E1 -29868.916,E2 -29868.916} C_VEL
LIN {X 0,Y 81.462,Z 536.666,A -85,B 0,C 180,E1 -29872.773,E2 -29872.773} C_VEL
LIN {X 0,Y 91.605,Z 532.389,A -85,B 0,C 180,E1 -29875.78,E2 -29875.78} C_VEL
LIN {X 0,Y 101.952,Z 526.85,A -85,B 0,C 180,E1 -29878.141,E2 -29878.141} C_VEL
LIN {X 0,Y 112.441,Z 519.867,A -85,B 0,C 180,E1 -29880.026,E2 -29880.026} C_VEL
LIN {X 0,Y 121.261,Z 512.678,A -85,B 0,C 180,E1 -29881.381,E2 -29881.381} C_VEL
LIN {X 0,Y 130.135,Z 503.941,A -85,B 0,C 180,E1 -29882.508,E2 -29882.508} C_VEL
LIN {X 0,Y 138.164,Z 494.254,A -85,B 0,C 180,E1 -29883.442,E2 -29883.442} C_VEL
LIN {X 0,Y 145.329,Z 483.629,A -85,B 0,C 180,E1 -29884.166,E2 -29884.166} C_VEL
LIN {X 0,Y 151.336,Z 472.477,A -85,B 0,C 180,E1 -29884.76,E2 -29884.76} C_VEL
LIN {X 0,Y 151.875,Z 471.32,A -85,B 0,C 180,E1 -29884.951,E2 -29884.951} C_VEL
LIN {X 0,Y 151.88,Z 471.354,A -85,B 0,C 180,E1 -29887.98,E2 -29887.98} C_VEL
LIN {X 0,Y 151.202,Z 472.955,A -85,B 0,C 180,E1 -29888.773,E2 -29888.773} C_VEL
LIN {X 0,Y 144.93,Z 484.521,A -85,B 0,C 180,E1 -29889.206,E2 -29889.206} C_VEL
LIN {X 0,Y 137.308,Z 495.704,A -85,B 0,C 180,E1 -29889.857,E2 -29889.857} C_VEL
LIN {X 0,Y 128.737,Z 505.782,A -85,B 0,C 180,E1 -29890.704,E2 -29890.704} C_VEL
LIN {X 0,Y 120.21,Z 514.029,A -85,B 0,C 180,E1 -29891.701,E2 -29891.701} C_VEL
LIN {X 0,Y 110.054,Z 522.121,A -85,B 0,C 180,E1 -29893.145,E2 -29893.145} C_VEL
LIN {X 0,Y 101.666,Z 527.648,A -85,B 0,C 180,E1 -29894.595,E2 -29894.595} C_VEL
LIN {X 0,Y 91.692,Z 533.075,A -85,B 0,C 180,E1 -29896.66,E2 -29896.66} C_VEL
LIN {X 0,Y 81.919,Z 537.343,A -85,B 0,C 180,E1 -29899.33,E2 -29899.33} C_VEL
LIN {X 0,Y 72.755,Z 540.487,A -85,B 0,C 180,E1 -29902.732,E2 -29902.732} C_VEL
LIN {X 0,Y 63.319,Z 542.865,A -85,B 0,C 180,E1 -29907.396,E2 -29907.396} C_VEL
LIN {X 0,Y 51.984,Z 544.521,A -85,B 0,C 180,E1 -29915.803,E2 -29915.803} C_VEL
LIN {X 0,Y 46.882,Z 544.786,A -85,B 0,C 180,E1 -29921.462,E2 -29921.462} C_VEL
LIN {X 0,Y 38.797,Z 544.111,A -85,B 0,C 180,E1 -29937.093,E2 -29937.093} C_VEL
LIN {X 0,Y 34.647,Z 541.913,A -85,B 0,C 180,E1 -29958.307,E2 -29958.307} C_VEL
LIN {X 0,Y 34.304,Z 540.177,A -85,B 0,C 180,E1 -29970.011,E2 -29970.011} C_VEL
LIN {X 0,Y 35.142,Z 536.653,A -85,B 0,C 180,E1 -29987.467,E2 -29987.467} C_VEL
LIN {X 0,Y 38.56,Z 531.976,A -85,B 0,C 180,E1 -30003.158,E2 -30003.158} C_VEL
LIN {X 0,Y 45.415,Z 524.9,A -85,B 0,C 180,E1 -30017.324,E2 -30017.324} C_VEL
LIN {X 0,Y 52.811,Z 517.199,A -85,B 0,C 180,E1 -30026.29,E2 -30026.29} C_VEL
LIN {X 0,Y 59.495,Z 509.521,A -85,B 0,C 180,E1 -30031.894,E2 -30031.894} C_VEL
LIN {X 0,Y 67.063,Z 499.598,A -85,B 0,C 180,E1 -30036.5,E2 -30036.5} C_VEL
LIN {X 0,Y 73.167,Z 490.123,A -85,B 0,C 180,E1 -30039.489,E2 -30039.489} C_VEL
LIN {X 0,Y 78.763,Z 480.06,A -85,B 0,C 180,E1 -30041.467,E2 -30041.467} C_VEL
LIN {X 0,Y 82.744,Z 471.192,A -85,B 0,C 180,E1 -30042.863,E2 -30042.863} C_VEL
LIN {X 0,Y 87.19,Z 458.659,A -85,B 0,C 180,E1 -30044.216,E2 -30044.216} C_VEL
LIN {X 0,Y 90.369,Z 445.929,A -85,B 0,C 180,E1 -30045.149,E2 -30045.149} C_VEL
LIN {X 0,Y 92.388,Z 432.443,A -85,B 0,C 180,E1 -30045.687,E2 -30045.687} C_VEL
LIN {X 0,Y 93.991,Z 417.262,A -85,B 0,C 180,E1 -30046.366,E2 -30046.366} C_VEL
LIN {X 0,Y 92.385,Z 412.343,A -85,B 0,C 180,E1 -30050.472,E2 -30050.472} C_VEL
LIN {X 0,Y 90.813,Z 407.799,A -85,B 0,C 180,E1 -30055.938,E2 -30055.938} C_VEL
LIN {X 0,Y 89.955,Z 404.805,A -85,B 0,C 180,E1 -30061.177,E2 -30061.177} C_VEL
LIN {X 0,Y 89.5,Z 404.607,A -85,B 0,C 180,E1 -30066.942,E2 -30066.942} C_VEL
LIN {X 0,Y 89.88,Z 405.234,A -85,B 0,C 180,E1 -30073.136,E2 -30073.136} C_VEL
LIN {X 0,Y 91.055,Z 408.942,A -85,B 0,C 180,E1 -30079.704,E2 -30079.704} C_VEL
LIN {X 0,Y 92.35,Z 412.327,A -85,B 0,C 180,E1 -30083.917,E2 -30083.917} C_VEL
LIN {X 0,Y 93.962,Z 417.16,A -85,B 0,C 180,E1 -30088.035,E2 -30088.035} C_VEL
LIN {X 0,Y 91.523,Z 438.157,A -85,B 0,C 180,E1 -30088.82,E2 -30088.82} C_VEL
LIN {X 0,Y 88.744,Z 451.617,A -85,B 0,C 180,E1 -30089.611,E2 -30089.611} C_VEL
LIN {X 0,Y 84.628,Z 464.873,A -85,B 0,C 180,E1 -30090.882,E2 -30090.882} C_VEL
LIN {X 0,Y 79.453,Z 477.273,A -85,B 0,C 180,E1 -30092.819,E2 -30092.819} C_VEL
LIN {X 0,Y 74.618,Z 486.524,A -85,B 0,C 180,E1 -30094.818,E2 -30094.818} C_VEL
LIN {X 0,Y 71.381,Z 491.378,A -85,B 0,C 180,E1 -30095.61,E2 -30095.61} C_VEL
LIN {X 0,Y 62.201,Z 501.781,A -85,B 0,C 180,E1 -30096.089,E2 -30096.089} C_VEL
LIN {X 0,Y 56.681,Z 507.381,A -85,B 0,C 180,E1 -30097.064,E2 -30097.064} C_VEL
LIN {X 0,Y 54.084,Z 510.067,A -85,B 0,C 180,E1 -30098.285,E2 -30098.285} C_VEL
LIN {X 0,Y 46.551,Z 517.726,A -85,B 0,C 180,E1 -30104.172,E2 -30104.172} C_VEL
LIN {X 0,Y 38.611,Z 525.003,A -85,B 0,C 180,E1 -30113.72,E2 -30113.72} C_VEL
LIN {X 0,Y 33.062,Z 529.91,A -85,B 0,C 180,E1 -30124.828,E2 -30124.828} C_VEL
LIN {X 0,Y 28.305,Z 534.778,A -85,B 0,C 180,E1 -30143.27,E2 -30143.27} C_VEL
LIN {X 0,Y 26.613,Z 538.382,A -85,B 0,C 180,E1 -30165.298,E2 -30165.298} C_VEL
LIN {X 0,Y 27.679,Z 540.266,A -85,B 0,C 180,E1 -30180.503,E2 -30180.503} C_VEL
LIN {X 0,Y 31.951,Z 542.176,A -85,B 0,C 180,E1 -30198.712,E2 -30198.712} C_VEL
LIN {X 0,Y 39.308,Z 543.295,A -85,B 0,C 180,E1 -30213.355,E2 -30213.355} C_VEL
LIN {X 0,Y 48.452,Z 543.346,A -85,B 0,C 180,E1 -30223.138,E2 -30223.138} C_VEL
LIN {X 0,Y 57.261,Z 542.486,A -85,B 0,C 180,E1 -30229.045,E2 -30229.045} C_VEL
LIN {X 0,Y 68.526,Z 540.32,A -85,B 0,C 180,E1 -30234.115,E2 -30234.115} C_VEL
LIN {X 0,Y 80.864,Z 536.544,A -85,B 0,C 180,E1 -30238,E2 -30238} C_VEL
LIN {X 0,Y 91.359,Z 532.169,A -85,B 0,C 180,E1 -30240.419,E2 -30240.419} C_VEL
LIN {X 0,Y 101.98,Z 526.525,A -85,B 0,C 180,E1 -30242.286,E2 -30242.286} C_VEL
LIN {X 0,Y 112.687,Z 519.412,A -85,B 0,C 180,E1 -30243.788,E2 -30243.788} C_VEL
LIN {X 0,Y 123.457,Z 510.403,A -85,B 0,C 180,E1 -30245.023,E2 -30245.023} C_VEL
LIN {X 0,Y 132.712,Z 500.839,A -85,B 0,C 180,E1 -30245.933,E2 -30245.933} C_VEL
LIN {X 0,Y 137.998,Z 494.297,A -85,B 0,C 180,E1 -30246.396,E2 -30246.396} C_VEL
LIN {X 0,Y 136.99,Z 495.672,A -85,B 0,C 180,E1 -30246.88,E2 -30246.88} C_VEL
LIN {X 0,Y 129.353,Z 504.652,A -85,B 0,C 180,E1 -30247.476,E2 -30247.476} C_VEL
LIN {X 0,Y 120.684,Z 513.075,A -85,B 0,C 180,E1 -30248.138,E2 -30248.138} C_VEL
LIN {X 0,Y 112.106,Z 520.057,A -85,B 0,C 180,E1 -30249.136,E2 -30249.136} C_VEL
LIN {X 0,Y 101.82,Z 526.929,A -85,B 0,C 180,E1 -30250.417,E2 -30250.417} C_VEL
LIN {X 0,Y 89.913,Z 533.266,A -85,B 0,C 180,E1 -30252.318,E2 -30252.318} C_VEL
LIN {X 0,Y 79.847,Z 537.444,A -85,B 0,C 180,E1 -30254.508,E2 -30254.508} C_VEL
LIN {X 0,Y 69.495,Z 540.731,A -85,B 0,C 180,E1 -30257.663,E2 -30257.663} C_VEL
LIN {X 0,Y 60.373,Z 542.802,A -85,B 0,C 180,E1 -30261.384,E2 -30261.384} C_VEL
LIN {X 0,Y 48.172,Z 544.381,A -85,B 0,C 180,E1 -30268.929,E2 -30268.929} C_VEL
LIN {X 0,Y 42.512,Z 544.581,A -85,B 0,C 180,E1 -30274.265,E2 -30274.265} C_VEL
LIN {X 0,Y 33.034,Z 543.815,A -85,B 0,C 180,E1 -30290.353,E2 -30290.353} C_VEL
LIN {X 0,Y 29.705,Z 542.87,A -85,B 0,C 180,E1 -30301.773,E2 -30301.773} C_VEL
LIN {X 0,Y 27.732,Z 541.53,A -85,B 0,C 180,E1 -30315.333,E2 -30315.333} C_VEL
LIN {X 0,Y 27.22,Z 539.723,A -85,B 0,C 180,E1 -30330.013,E2 -30330.013} C_VEL
LIN {X 0,Y 28.428,Z 536.109,A -85,B 0,C 180,E1 -30351.781,E2 -30351.781} C_VEL
LIN {X 0,Y 32.81,Z 531.337,A -85,B 0,C 180,E1 -30370.001,E2 -30370.001} C_VEL
LIN {X 0,Y 39.617,Z 525.287,A -85,B 0,C 180,E1 -30382.983,E2 -30382.983} C_VEL
LIN {X 0,Y 47.748,Z 517.718,A -85,B 0,C 180,E1 -30392.037,E2 -30392.037} C_VEL
LIN {X 0,Y 54.985,Z 510.131,A -85,B 0,C 180,E1 -30397.451,E2 -30397.451} C_VEL
LIN {X 0,Y 62.153,Z 501.564,A -85,B 0,C 180,E1 -30401.281,E2 -30401.281} C_VEL
LIN {X 0,Y 68.522,Z 492.541,A -85,B 0,C 180,E1 -30404.078,E2 -30404.078} C_VEL
LIN {X 0,Y 75.137,Z 481.518,A -85,B 0,C 180,E1 -30406.052,E2 -30406.052} C_VEL
LIN {X 0,Y 80.094,Z 471.069,A -85,B 0,C 180,E1 -30407.49,E2 -30407.49} C_VEL
LIN {X 0,Y 84.684,Z 458.559,A -85,B 0,C 180,E1 -30408.636,E2 -30408.636} C_VEL
LIN {X 0,Y 88.07,Z 445.371,A -85,B 0,C 180,E1 -30409.446,E2 -30409.446} C_VEL
LIN {X 0,Y 90.251,Z 430.691,A -85,B 0,C 180,E1 -30409.942,E2 -30409.942} C_VEL
LIN {X 0,Y 91.356,Z 420.764,A -85,B 0,C 180,E1 -30410.333,E2 -30410.333} C_VEL
LIN {X 0,Y 90.022,Z 416.134,A -85,B 0,C 180,E1 -30415.101,E2 -30415.101} C_VEL
LIN {X 0,Y 89.293,Z 413.614,A -85,B 0,C 180,E1 -30418.871,E2 -30418.871} C_VEL
LIN {X 0,Y 88.932,Z 411.71,A -85,B 0,C 180,E1 -30422.263,E2 -30422.263} C_VEL
LIN {X 0,Y 88.66,Z 411.752,A -85,B 0,C 180,E1 -30429.121,E2 -30429.121} C_VEL
LIN {X 0,Y 88.886,Z 412.33,A -85,B 0,C 180,E1 -30432.417,E2 -30432.417} C_VEL
LIN {X 0,Y 89.745,Z 415.559,A -85,B 0,C 180,E1 -30438.254,E2 -30438.254} C_VEL
LIN {X 0,Y 90.804,Z 418.857,A -85,B 0,C 180,E1 -30442.36,E2 -30442.36} C_VEL
LIN {X 0,Y 91.318,Z 420.753,A -85,B 0,C 180,E1 -30444.05,E2 -30444.05} C_VEL
LIN {X 0,Y 88.626,Z 441.334,A -85,B 0,C 180,E1 -30444.692,E2 -30444.692} C_VEL
LIN {X 0,Y 85.631,Z 454.32,A -85,B 0,C 180,E1 -30445.462,E2 -30445.462} C_VEL
LIN {X 0,Y 81.371,Z 466.804,A -85,B 0,C 180,E1 -30446.533,E2 -30446.533} C_VEL
LIN {X 0,Y 75.853,Z 479.071,A -85,B 0,C 180,E1 -30448.324,E2 -30448.324} C_VEL
LIN {X 0,Y 69.337,Z 490.381,A -85,B 0,C 180,E1 -30450.586,E2 -30450.586} C_VEL
LIN {X 0,Y 63.055,Z 499.378,A -85,B 0,C 180,E1 -30453.277,E2 -30453.277} C_VEL
LIN {X 0,Y 55.368,Z 508.682,A -85,B 0,C 180,E1 -30457.493,E2 -30457.493} C_VEL
LIN {X 0,Y 54.084,Z 510.067,A -85,B 0,C 180,E1 -30458.285,E2 -30458.285} C_VEL
LIN {X 0,Y 50.02,Z 513.978,A -85,B 0,C 180,E1 -30460.244,E2 -30460.244} C_VEL
LIN {X 0,Y 42.273,Z 519.852,A -85,B 0,C 180,E1 -30462.606,E2 -30462.606} C_VEL
LIN {X 0,Y 34.265,Z 525.19,A -85,B 0,C 180,E1 -30466.399,E2 -30466.399} C_VEL
LIN {X 0,Y 29.996,Z 528.101,A -85,B 0,C 180,E1 -30471.437,E2 -30471.437} C_VEL
LIN {X 0,Y 22.71,Z 533.804,A -85,B 0,C 180,E1 -30491.956,E2 -30491.956} C_VEL
LIN {X 0,Y 19.57,Z 537.757,A -85,B 0,C 180,E1 -30520.325,E2 -30520.325} C_VEL
LIN {X 0,Y 21.672,Z 540.662,A -85,B 0,C 180,E1 -30550.413,E2 -30550.413} C_VEL
LIN {X 0,Y 26.775,Z 542.326,A -85,B 0,C 180,E1 -30568.338,E2 -30568.338} C_VEL
LIN {X 0,Y 36.579,Z 543.532,A -85,B 0,C 180,E1 -30583.839,E2 -30583.839} C_VEL
LIN {X 0,Y 45.638,Z 543.565,A -85,B 0,C 180,E1 -30591.144,E2 -30591.144} C_VEL
LIN {X 0,Y 56.322,Z 542.58,A -85,B 0,C 180,E1 -30596.509,E2 -30596.509} C_VEL
LIN {X 0,Y 66.918,Z 540.605,A -85,B 0,C 180,E1 -30600.001,E2 -30600.001} C_VEL
LIN {X 0,Y 77.378,Z 537.676,A -85,B 0,C 180,E1 -30602.561,E2 -30602.561} C_VEL
LIN {X 0,Y 89.59,Z 532.924,A -85,B 0,C 180,E1 -30604.741,E2 -30604.741} C_VEL
LIN {X 0,Y 98.929,Z 528.267,A -85,B 0,C 180,E1 -30606.01,E2 -30606.01} C_VEL
LIN {X 0,Y 99.049,Z 528.222,A -85,B 0,C 180,E1 -30606.641,E2 -30606.641} C_VEL
LIN {X 0,Y 88.052,Z 533.742,A -85,B 0,C 180,E1 -30607.914,E2 -30607.914} C_VEL
LIN {X 0,Y 78.371,Z 537.545,A -85,B 0,C 180,E1 -30609.479,E2 -30609.479} C_VEL
LIN {X 0,Y 66.622,Z 541.021,A -85,B 0,C 180,E1 -30612.181,E2 -30612.181} C_VEL
LIN {X 0,Y 58.157,Z 542.739,A -85,B 0,C 180,E1 -30614.839,E2 -30614.839} C_VEL
LIN {X 0,Y 45.159,Z 544.227,A -85,B 0,C 180,E1 -30620.993,E2 -30620.993} C_VEL
LIN {X 0,Y 33.111,Z 544.124,A -85,B 0,C 180,E1 -30631.915,E2 -30631.915} C_VEL
LIN {X 0,Y 23.676,Z 542.535,A -85,B 0,C 180,E1 -30653.6,E2 -30653.6} C_VEL
LIN {X 0,Y 20.931,Z 541.12,A -85,B 0,C 180,E1 -30670.399,E2 -30670.399} C_VEL
LIN {X 0,Y 20.114,Z 539.266,A -85,B 0,C 180,E1 -30690.018,E2 -30690.018} C_VEL
LIN {X 0,Y 21.983,Z 535.566,A -85,B 0,C 180,E1 -30718.675,E2 -30718.675} C_VEL
LIN {X 0,Y 27.709,Z 530.696,A -85,B 0,C 180,E1 -30739.564,E2 -30739.564} C_VEL
LIN {X 0,Y 35.776,Z 524.545,A -85,B 0,C 180,E1 -30752.151,E2 -30752.151} C_VEL
LIN {X 0,Y 44.837,Z 516.854,A -85,B 0,C 180,E1 -30760.154,E2 -30760.154} C_VEL
LIN {X 0,Y 51.855,Z 509.956,A -85,B 0,C 180,E1 -30764.27,E2 -30764.27} C_VEL
LIN {X 0,Y 59.407,Z 501.403,A -85,B 0,C 180,E1 -30767.446,E2 -30767.446} C_VEL
LIN {X 0,Y 66.069,Z 492.386,A -85,B 0,C 180,E1 -30769.753,E2 -30769.753} C_VEL
LIN {X 0,Y 72.89,Z 481.381,A -85,B 0,C 180,E1 -30771.256,E2 -30771.256} C_VEL
LIN {X 0,Y 77.998,Z 470.943,A -85,B 0,C 180,E1 -30772.407,E2 -30772.407} C_VEL
LIN {X 0,Y 82.866,Z 457.978,A -85,B 0,C 180,E1 -30773.332,E2 -30773.332} C_VEL
LIN {X 0,Y 86.1,Z 445.724,A -85,B 0,C 180,E1 -30773.931,E2 -30773.931} C_VEL
LIN {X 0,Y 88.249,Z 432.177,A -85,B 0,C 180,E1 -30774.296,E2 -30774.296} C_VEL
LIN {X 0,Y 89.11,Z 424.504,A -85,B 0,C 180,E1 -30774.641,E2 -30774.641} C_VEL
LIN {X 0,Y 88.28,Z 420.705,A -85,B 0,C 180,E1 -30779.429,E2 -30779.429} C_VEL
LIN {X 0,Y 87.928,Z 418.675,A -85,B 0,C 180,E1 -30783.436,E2 -30783.436} C_VEL
LIN {X 0,Y 87.887,Z 419.029,A -85,B 0,C 180,E1 -30791.024,E2 -30791.024} C_VEL
LIN {X 0,Y 88.468,Z 422.049,A -85,B 0,C 180,E1 -30796.592,E2 -30796.592} C_VEL
LIN {X 0,Y 89.083,Z 424.442,A -85,B 0,C 180,E1 -30799.721,E2 -30799.721} C_VEL
LIN {X 0,Y 86.476,Z 443.104,A -85,B 0,C 180,E1 -30800.306,E2 -30800.306} C_VEL
LIN {X 0,Y 83.585,Z 454.886,A -85,B 0,C 180,E1 -30800.882,E2 -30800.882} C_VEL
LIN {X 0,Y 79.412,Z 466.757,A -85,B 0,C 180,E1 -30801.67,E2 -30801.67} C_VEL
LIN {X 0,Y 73.588,Z 479.289,A -85,B 0,C 180,E1 -30803.175,E2 -30803.175} C_VEL
LIN {X 0,Y 66.946,Z 490.416,A -85,B 0,C 180,E1 -30804.963,E2 -30804.963} C_VEL
LIN {X 0,Y 59.445,Z 500.594,A -85,B 0,C 180,E1 -30807.526,E2 -30807.526} C_VEL
LIN {X 0,Y 50.888,Z 510.169,A -85,B 0,C 180,E1 -30811.384,E2 -30811.384} C_VEL
LIN {X 0,Y 41.885,Z 518.619,A -85,B 0,C 180,E1 -30817.14,E2 -30817.14} C_VEL
LIN {X 0,Y 33.133,Z 525.734,A -85,B 0,C 180,E1 -30826.404,E2 -30826.404} C_VEL
LIN {X 0,Y 29.996,Z 528.101,A -85,B 0,C 180,E1 -30831.437,E2 -30831.437} C_VEL
LIN {X 0,Y 25.893,Z 530.869,A -85,B 0,C 180,E1 -30838.106,E2 -30838.106} C_VEL
LIN {X 0,Y 18.489,Z 534.822,A -85,B 0,C 180,E1 -30852.065,E2 -30852.065} C_VEL
LIN {X 0,Y 13.719,Z 537.417,A -85,B 0,C 180,E1 -30873.427,E2 -30873.427} C_VEL
LIN {X 0,Y 12.867,Z 539.051,A -85,B 0,C 180,E1 -30898.144,E2 -30898.144} C_VEL
LIN {X 0,Y 13.376,Z 539.534,A -85,B 0,C 180,E1 -30906.297,E2 -30906.297} C_VEL
LIN {X 0,Y 16.771,Z 541.057,A -85,B 0,C 180,E1 -30926.901,E2 -30926.901} C_VEL
LIN {X 0,Y 22.631,Z 542.465,A -85,B 0,C 180,E1 -30941.913,E2 -30941.913} C_VEL
LIN {X 0,Y 28.54,Z 543.308,A -85,B 0,C 180,E1 -30949.987,E2 -30949.987} C_VEL
LIN {X 0,Y 35.241,Z 543.761,A -85,B 0,C 180,E1 -30955.518,E2 -30955.518} C_VEL
LIN {X 0,Y 43.785,Z 543.779,A -85,B 0,C 180,E1 -30960.002,E2 -30960.002} C_VEL
LIN {X 0,Y 56.361,Z 542.644,A -85,B 0,C 180,E1 -30964.087,E2 -30964.087} C_VEL
LIN {X 0,Y 63.554,Z 541.392,A -85,B 0,C 180,E1 -30965.651,E2 -30965.651} C_VEL
LIN {X 0,Y 64.43,Z 541.227,A -85,B 0,C 180,E1 -30966.264,E2 -30966.264} C_VEL
LIN {X 0,Y 56.753,Z 542.676,A -85,B 0,C 180,E1 -30967.879,E2 -30967.879} C_VEL
LIN {X 0,Y 49.897,Z 543.571,A -85,B 0,C 180,E1 -30969.663,E2 -30969.663} C_VEL
LIN {X 0,Y 36.457,Z 544.145,A -85,B 0,C 180,E1 -30975.485,E2 -30975.485} C_VEL
LIN {X 0,Y 23.863,Z 543.223,A -85,B 0,C 180,E1 -30987.961,E2 -30987.961} C_VEL
LIN {X 0,Y 18.443,Z 542.18,A -85,B 0,C 180,E1 -31000.38,E2 -31000.38} C_VEL
LIN {X 0,Y 14.442,Z 540.705,A -85,B 0,C 180,E1 -31020.91,E2 -31020.91} C_VEL
LIN {X 0,Y 13.009,Z 538.811,A -85,B 0,C 180,E1 -31050.028,E2 -31050.028} C_VEL
LIN {X 0,Y 16.089,Z 535.021,A -85,B 0,C 180,E1 -31090.967,E2 -31090.967} C_VEL
LIN {X 0,Y 23.702,Z 530.056,A -85,B 0,C 180,E1 -31112.849,E2 -31112.849} C_VEL
LIN {X 0,Y 33.04,Z 523.801,A -85,B 0,C 180,E1 -31123.214,E2 -31123.214} C_VEL
LIN {X 0,Y 42.932,Z 515.942,A -85,B 0,C 180,E1 -31129.217,E2 -31129.217} C_VEL
LIN {X 0,Y 51.409,Z 507.89,A -85,B 0,C 180,E1 -31132.411,E2 -31132.411} C_VEL
LIN {X 0,Y 60.006,Z 498.057,A -85,B 0,C 180,E1 -31134.646,E2 -31134.646} C_VEL
LIN {X 0,Y 66.05,Z 489.677,A -85,B 0,C 180,E1 -31136.056,E2 -31136.056} C_VEL
LIN {X 0,Y 72.15,Z 479.644,A -85,B 0,C 180,E1 -31136.877,E2 -31136.877} C_VEL
LIN {X 0,Y 76.505,Z 470.82,A -85,B 0,C 180,E1 -31137.546,E2 -31137.546} C_VEL
LIN {X 0,Y 81.361,Z 458.201,A -85,B 0,C 180,E1 -31138.16,E2 -31138.16} C_VEL
LIN {X 0,Y 84.856,Z 445.255,A -85,B 0,C 180,E1 -31138.604,E2 -31138.604} C_VEL
LIN {X 0,Y 87.184,Z 430.322,A -85,B 0,C 180,E1 -31138.89,E2 -31138.89} C_VEL
LIN {X 0,Y 87.351,Z 428.687,A -85,B 0,C 180,E1 -31139.07,E2 -31139.07} C_VEL
LIN {X 0,Y 87.002,Z 425.844,A -85,B 0,C 180,E1 -31143.762,E2 -31143.762} C_VEL
LIN {X 0,Y 86.872,Z 425.735,A -85,B 0,C 180,E1 -31146.928,E2 -31146.928} C_VEL
LIN {X 0,Y 86.945,Z 426.134,A -85,B 0,C 180,E1 -31150.406,E2 -31150.406} C_VEL
